C05447=1098.958,349.273,-87.589,179.031,19.110,152.319
C05448=1098.953,349.026,-87.554,179.028,19.106,152.319
C05449=1098.947,348.778,-87.521,179.025,19.103,152.319
C05450=1098.941,348.529,-87.486,179.022,19.099,152.318
C05451=1098.935,348.282,-87.452,179.019,19.095,152.318
C05452=1098.930,348.035,-87.418,179.016,19.092,152.318
C05453=1098.924,347.787,-87.385,179.013,19.089,152.318
C05454=1098.918,347.540,-87.351,179.010,19.084,152.317
C05455=1098.913,347.292,-87.316,179.007,19.081,152.317
C05456=1098.907,347.044,-87.283,179.003,19.078,152.317
C05457=1098.902,346.797,-87.249,179.000,19.074,152.316
C05458=1098.895,346.549,-87.214,178.998,19.071,152.316
C05459=1098.890,346.301,-87.181,178.994,19.067,152.316
C05460=1098.884,346.054,-87.147,178.992,19.064,152.316
C05461=1098.879,345.806,-87.112,178.988,19.060,152.315
C05462=1098.873,345.558,-87.079,178.985,19.057,152.315
C05463=1098.867,345.311,-87.045,178.982,19.053,152.315
C05464=1098.862,345.063,-87.011,178.979,19.050,152.314
C05465=1098.856,344.816,-86.977,178.976,19.046,152.314
C05466=1098.850,344.568,-86.944,178.973,19.043,152.314
C05467=1098.844,344.320,-86.910,178.969,19.039,152.314
C05468=1098.839,344.073,-86.877,178.966,19.036,152.313
C05469=1098.829,343.698,-86.825,178.962,19.031,152.313
C05470=1098.821,343.324,-86.774,178.957,19.026,152.313
C05471=1098.812,342.950,-86.724,178.952,19.021,152.312
C05472=1098.804,342.576,-86.673,178.947,19.015,152.312
C05473=1098.798,342.328,-86.640,178.945,19.012,152.312
C05474=1098.793,342.080,-86.606,178.941,19.008,152.311
C05475=1098.787,341.833,-86.572,178.938,19.006,152.311
C05476=1098.781,341.585,-86.539,178.935,19.003,152.311
C05477=1098.776,341.337,-86.505,178.932,18.999,152.311
C05478=1098.770,341.089,-86.472,178.929,18.996,152.311
C05479=1098.764,340.842,-86.438,178.925,18.992,152.310
C05480=1098.759,340.594,-86.404,178.923,18.989,152.310
C05481=1098.753,340.346,-86.371,178.920,18.986,152.310
C05482=1098.747,340.099,-86.338,178.916,18.982,152.310
C05483=1098.741,339.851,-86.305,178.913,18.979,152.310
C05484=1098.736,339.603,-86.271,178.910,18.975,152.309
C05485=1098.730,339.356,-86.237,178.907,18.972,152.309
C05486=1098.724,339.108,-86.204,178.904,18.970,152.309
C05487=1098.719,338.860,-86.171,178.901,18.966,152.309
C05488=1098.713,338.612,-86.137,178.898,18.963,152.308
C05489=1098.707,338.364,-86.105,178.895,18.960,152.308
C05490=1098.701,338.116,-86.071,178.891,18.956,152.308
C05491=1098.696,337.869,-86.038,178.888,18.953,152.308
C05492=1098.690,337.621,-86.004,178.885,18.950,152.308
C05493=1098.684,337.374,-85.971,178.882,18.947,152.308
C05494=1098.678,337.126,-85.938,178.879,18.944,152.307
C05495=1098.672,336.878,-85.904,178.875,18.940,152.307
C05496=1098.667,336.630,-85.871,178.872,18.937,152.307
C05497=1098.661,336.382,-85.838,178.870,18.934,152.307
C05498=1098.656,336.135,-85.805,178.866,18.931,152.307
C05499=1098.650,335.887,-85.772,178.863,18.928,152.306
C05500=1098.644,335.640,-85.739,178.860,18.925,152.306
C05501=1098.638,335.392,-85.706,178.856,18.921,152.306
C05502=1098.633,335.144,-85.673,178.853,18.919,152.306
C05503=1098.627,334.896,-85.641,178.851,18.915,152.306
C05504=1098.621,334.648,-85.607,178.848,18.913,152.306
C05505=1098.616,334.400,-85.574,178.844,18.909,152.305
C05506=1098.610,334.153,-85.542,178.841,18.906,152.305
C05507=1098.604,333.905,-85.508,178.838,18.903,152.305
C05508=1098.599,333.657,-85.475,178.834,18.900,152.305
C05509=1098.593,333.410,-85.442,178.831,18.897,152.305
C05510=1098.587,333.161,-85.410,178.829,18.894,152.305
C05511=1098.582,332.913,-85.376,178.825,18.891,152.305
C05512=1098.576,332.666,-85.344,178.822,18.888,152.304
C05513=1098.570,332.418,-85.311,178.819,18.885,152.304
C05514=1098.564,332.170,-85.278,178.815,18.881,152.304
C05515=1098.559,331.922,-85.245,178.812,18.879,152.304
C05516=1098.553,331.675,-85.212,178.809,18.876,152.304
C05517=1098.547,331.427,-85.179,178.806,18.873,152.304
C05518=1098.542,331.179,-85.147,178.803,18.870,152.304
C05519=1098.535,330.932,-85.115,178.800,18.867,152.304
C05520=1098.530,330.684,-85.081,178.797,18.864,152.303
C05521=1098.520,330.303,-85.031,178.791,18.859,152.303
C05522=1098.511,329.923,-84.981,178.787,18.855,152.303
C05523=1098.504,329.542,-84.932,178.781,18.851,152.303
C05524=1098.494,329.162,-84.881,178.777,18.846,152.303
C05525=1098.488,328.915,-84.849,178.774,18.844,152.303
C05526=1098.483,328.666,-84.816,178.770,18.840,152.303
C05527=1098.477,328.419,-84.784,178.767,18.838,152.303
C05528=1098.471,328.170,-84.752,178.764,18.835,152.303
C05529=1098.465,327.923,-84.719,178.761,18.832,152.302
C05530=1098.460,327.675,-84.687,178.757,18.829,152.302
C05531=1098.454,327.427,-84.654,178.754,18.826,152.302
C05532=1098.448,327.179,-84.622,178.751,18.823,152.302
C05533=1098.442,326.931,-84.589,178.748,18.821,152.302
C05534=1098.437,326.684,-84.557,178.745,18.818,152.302
C05535=1098.430,326.436,-84.524,178.742,18.815,152.302
C05536=1098.424,326.188,-84.492,178.738,18.812,152.302
C05537=1098.420,325.940,-84.460,178.735,18.810,152.302
C05538=1098.413,325.693,-84.427,178.732,18.807,152.302
C05539=1098.407,325.444,-84.395,178.729,18.803,152.302
C05540=1098.402,325.197,-84.363,178.726,18.801,152.302
C05541=1098.397,324.949,-84.330,178.723,18.798,152.301
C05542=1098.391,324.701,-84.298,178.720,18.795,152.301
C05543=1098.385,324.453,-84.266,178.717,18.793,152.301
C05544=1098.379,324.206,-84.234,178.713,18.790,152.301
C05545=1098.374,323.957,-84.201,178.710,18.787,152.301
C05546=1098.368,323.710,-84.169,178.707,18.784,152.301
C05547=1098.362,323.461,-84.137,178.704,18.781,152.301
C05548=1098.356,323.214,-84.105,178.701,18.779,152.301
C05549=1098.351,322.966,-84.073,178.698,18.776,152.301
C05550=1098.345,322.718,-84.040,178.693,18.773,152.301
C05551=1098.340,322.470,-84.009,178.690,18.770,152.301
C05552=1098.334,322.222,-83.977,178.687,18.768,152.301
C05553=1098.329,322.012,-83.950,178.684,18.765,152.301
C05554=1098.324,321.802,-83.922,178.682,18.763,152.301
C05555=1098.320,321.592,-83.895,178.679,18.760,152.301
C05556=1098.315,321.381,-83.868,178.677,18.759,152.301
C05557=1098.310,321.171,-83.841,178.674,18.756,152.301
C05558=1098.306,320.961,-83.814,178.671,18.754,152.300
C05559=1098.301,320.751,-83.787,178.668,18.752,152.301
C05560=1098.296,320.541,-83.760,178.666,18.749,152.300
C05561=1098.290,320.293,-83.728,178.663,18.747,152.300
C05562=1098.285,320.045,-83.696,178.659,18.744,152.300
C05563=1098.279,319.797,-83.664,178.656,18.741,152.300
C05564=1098.273,319.549,-83.632,178.653,18.738,152.300
C05565=1098.267,319.301,-83.600,178.650,18.736,152.300
C05566=1098.262,319.054,-83.568,178.647,18.733,152.300
C05567=1098.256,318.805,-83.536,178.644,18.731,152.300
C05568=1098.251,318.558,-83.505,178.640,18.728,152.300
C05569=1098.245,318.310,-83.473,178.637,18.725,152.300
C05570=1098.239,318.062,-83.441,178.634,18.722,152.300
C05571=1098.234,317.814,-83.408,178.630,18.720,152.300
C05572=1098.229,317.566,-83.377,178.627,18.717,152.300
C05573=1098.223,317.334,-83.348,178.624,18.715,152.300
C05574=1098.218,317.104,-83.318,178.621,18.712,152.300
C05575=1098.213,316.872,-83.288,178.618,18.709,152.300
C05576=1098.207,316.640,-83.259,178.616,18.708,152.300
C05577=1098.203,316.409,-83.229,178.613,18.705,152.300
C05578=1098.198,316.177,-83.200,178.609,18.703,152.300
C05579=1098.191,315.946,-83.170,178.606,18.700,152.300
C05580=1098.187,315.715,-83.141,178.603,18.698,152.300
C05581=1098.181,315.467,-83.109,178.600,18.695,152.300
C05582=1098.176,315.219,-83.077,178.597,18.692,152.300
C05583=1098.170,314.971,-83.045,178.594,18.690,152.300
C05584=1098.164,314.723,-83.014,178.591,18.687,152.300
C05585=1098.158,314.475,-82.983,178.587,18.685,152.300
C05586=1098.152,314.227,-82.951,178.584,18.682,152.300
C05587=1098.147,313.979,-82.920,178.581,18.680,152.300
C05588=1098.141,313.731,-82.889,178.578,18.678,152.300
C05589=1098.135,313.484,-82.857,178.574,18.675,152.300
C05590=1098.129,313.235,-82.826,178.571,18.673,152.300
C05591=1098.123,312.988,-82.795,178.568,18.670,152.300
C05592=1098.117,312.740,-82.763,178.564,18.668,152.300
C05593=1098.112,312.492,-82.732,178.561,18.665,152.300
C05594=1098.106,312.244,-82.700,178.558,18.663,152.300
C05595=1098.100,311.995,-82.669,178.555,18.661,152.300
C05596=1098.095,311.748,-82.638,178.552,18.658,152.300
C05597=1098.089,311.499,-82.607,178.548,18.656,152.300
C05598=1098.083,311.252,-82.575,178.545,18.653,152.300
C05599=1098.077,311.004,-82.544,178.542,18.651,152.300
C05600=1098.072,310.756,-82.513,178.539,18.649,152.300
C05601=1098.066,310.508,-82.481,178.535,18.646,152.300
C05602=1098.060,310.260,-82.451,178.532,18.644,152.300
C05603=1098.055,310.012,-82.420,178.528,18.641,152.300
C05604=1098.048,309.765,-82.389,178.525,18.639,152.300
C05605=1098.043,309.516,-82.357,178.522,18.636,152.300
C05606=1098.037,309.268,-82.326,178.519,18.634,152.301
C05607=1098.032,309.020,-82.295,178.515,18.632,152.301
C05608=1098.026,308.773,-82.264,178.512,18.629,152.301
C05609=1098.020,308.524,-82.233,178.509,18.627,152.301
C05610=1098.015,308.276,-82.202,178.506,18.624,152.301
C05611=1098.009,308.029,-82.171,178.503,18.622,152.301
C05612=1098.003,307.780,-82.140,178.499,18.620,152.301
C05613=1097.997,307.532,-82.109,178.496,18.617,152.301
C05614=1097.992,307.285,-82.078,178.493,18.615,152.301
C05615=1097.986,307.037,-82.047,178.490,18.613,152.301
C05616=1097.980,306.788,-82.016,178.486,18.610,152.301
C05617=1097.974,306.540,-81.986,178.483,18.608,152.301
C05618=1097.969,306.293,-81.954,178.480,18.606,152.301
C05619=1097.963,306.045,-81.924,178.477,18.604,152.301
C05620=1097.958,305.797,-81.893,178.473,18.601,152.301
C05621=1097.952,305.548,-81.862,178.470,18.599,152.301
C05622=1097.946,305.301,-81.830,178.467,18.597,152.301
C05623=1097.941,305.053,-81.800,178.464,18.594,152.301
C05624=1097.935,304.805,-81.769,178.460,18.592,152.302
C05625=1097.930,304.557,-81.739,178.457,18.590,152.302
C05626=1097.924,304.308,-81.707,178.453,18.587,152.302
C05627=1097.918,304.060,-81.677,178.450,18.585,152.302
C05628=1097.912,303.813,-81.647,178.447,18.582,152.302
C05629=1097.904,303.428,-81.598,178.442,18.579,152.302
C05630=1097.895,303.043,-81.551,178.437,18.575,152.302
C05631=1097.887,302.658,-81.503,178.432,18.572,152.302
C05632=1097.878,302.274,-81.455,178.427,18.568,152.302
C05633=1097.872,302.026,-81.425,178.424,18.566,152.302
C05634=1097.867,301.778,-81.394,178.421,18.564,152.302
C05635=1097.861,301.530,-81.364,178.417,18.562,152.302
C05636=1097.855,301.282,-81.334,178.414,18.559,152.302
C05637=1097.850,301.034,-81.303,178.411,18.557,152.303
C05638=1097.845,300.786,-81.273,178.408,18.555,152.303
C05639=1097.839,300.538,-81.242,178.404,18.552,152.303
C05640=1097.834,300.290,-81.211,178.401,18.550,152.303
C05641=1097.827,300.041,-81.181,178.398,18.548,152.303
C05642=1097.821,299.793,-81.150,178.395,18.545,152.303
C05643=1097.816,299.545,-81.119,178.391,18.543,152.303
C05644=1097.811,299.298,-81.089,178.388,18.541,152.303
C05645=1097.805,299.049,-81.059,178.385,18.539,152.303
C05646=1097.800,298.801,-81.028,178.381,18.537,152.303
C05647=1097.794,298.553,-80.998,178.378,18.534,152.303
C05648=1097.788,298.305,-80.968,178.375,18.532,152.303
C05649=1097.782,298.057,-80.937,178.372,18.530,152.303
C05650=1097.778,297.809,-80.907,178.368,18.527,152.304
C05651=1097.772,297.561,-80.877,178.365,18.526,152.304
C05652=1097.766,297.313,-80.846,178.362,18.523,152.304
C05653=1097.761,297.065,-80.817,178.358,18.521,152.304
C05654=1097.755,296.817,-80.787,178.355,18.519,152.304
C05655=1097.749,296.569,-80.756,178.352,18.517,152.304
C05656=1097.743,296.321,-80.726,178.348,18.515,152.304
C05657=1097.738,296.073,-80.696,178.345,18.512,152.304
C05658=1097.732,295.825,-80.666,178.342,18.510,152.305
C05659=1097.727,295.576,-80.636,178.338,18.508,152.305
C05660=1097.721,295.328,-80.605,178.335,18.506,152.305
C05661=1097.715,295.081,-80.575,178.332,18.504,152.305
C05662=1097.710,294.832,-80.545,178.328,18.502,152.305
C05663=1097.704,294.584,-80.515,178.325,18.499,152.305
C05664=1097.699,294.336,-80.485,178.322,18.498,152.305
C05665=1097.693,294.088,-80.455,178.319,18.496,152.305
C05666=1097.687,293.840,-80.425,178.316,18.494,152.306
C05667=1097.681,293.592,-80.395,178.312,18.492,152.306
C05668=1097.676,293.344,-80.365,178.309,18.489,152.306
C05669=1097.670,293.095,-80.335,178.306,18.487,152.306
C05670=1097.665,292.847,-80.305,178.302,18.485,152.306
C05671=1097.659,292.599,-80.275,178.299,18.483,152.306
C05672=1097.652,292.351,-80.246,178.296,18.481,152.306
C05673=1097.647,292.103,-80.216,178.292,18.479,152.306
C05674=1097.641,291.855,-80.186,178.289,18.477,152.307
C05675=1097.635,291.607,-80.156,178.286,18.474,152.307
C05676=1097.630,291.359,-80.126,178.283,18.473,152.307
C05677=1097.625,291.111,-80.097,178.280,18.471,152.307
C05678=1097.619,290.863,-80.066,178.276,18.469,152.307
C05679=1097.614,290.615,-80.037,178.273,18.467,152.307
C05680=1097.608,290.366,-80.007,178.269,18.465,152.307
C05681=1097.600,289.996,-79.963,178.264,18.461,152.308
C05682=1097.590,289.625,-79.918,178.259,18.458,152.308
C05683=1097.582,289.254,-79.874,178.255,18.456,152.308
C05684=1097.574,288.883,-79.829,178.250,18.453,152.308
C05685=1097.568,288.635,-79.800,178.247,18.451,152.308
C05686=1097.562,288.386,-79.771,178.243,18.449,152.309
C05687=1097.557,288.139,-79.740,178.240,18.447,152.309
C05688=1097.551,287.890,-79.711,178.236,18.445,152.309
C05689=1097.545,287.642,-79.682,178.233,18.443,152.309
C05690=1097.539,287.394,-79.652,178.230,18.441,152.309
C05691=1097.534,287.145,-79.622,178.227,18.439,152.309
C05692=1097.528,286.898,-79.594,178.224,18.437,152.310
C05693=1097.522,286.650,-79.563,178.220,18.435,152.310
C05694=1097.517,286.402,-79.534,178.217,18.433,152.310
C05695=1097.511,286.153,-79.504,178.213,18.431,152.310
C05696=1097.505,285.905,-79.475,178.210,18.429,152.310
C05697=1097.500,285.657,-79.445,178.207,18.427,152.310
C05698=1097.495,285.409,-79.416,178.204,18.425,152.311
C05699=1097.488,285.161,-79.387,178.200,18.424,152.311
C05700=1097.483,284.912,-79.357,178.197,18.421,152.311
C05701=1097.477,284.664,-79.328,178.194,18.419,152.311
C05702=1097.471,284.416,-79.299,178.190,18.418,152.311
C05703=1097.466,284.168,-79.269,178.187,18.415,152.311
C05704=1097.461,283.919,-79.240,178.183,18.413,152.312
C05705=1097.455,283.671,-79.211,178.181,18.412,152.312
C05706=1097.449,283.423,-79.181,178.177,18.410,152.312
C05707=1097.443,283.175,-79.152,178.174,18.408,152.312
C05708=1097.438,282.927,-79.123,178.171,18.406,152.312
C05709=1097.432,282.679,-79.093,178.167,18.404,152.312
C05710=1097.426,282.430,-79.065,178.164,18.402,152.313
C05711=1097.422,282.182,-79.036,178.161,18.400,152.313
C05712=1097.415,281.934,-79.007,178.158,18.398,152.313
C05713=1097.410,281.685,-78.977,178.154,18.397,152.313
C05714=1097.405,281.438,-78.948,178.151,18.394,152.313
C05715=1097.399,281.190,-78.919,178.147,18.392,152.313
C05716=1097.393,280.941,-78.890,178.144,18.391,152.314
C05717=1097.387,280.692,-78.861,178.142,18.389,152.314
C05718=1097.382,280.445,-78.831,178.138,18.387,152.314
C05719=1097.376,280.197,-78.802,178.134,18.385,152.314
C05720=1097.370,279.948,-78.774,178.131,18.383,152.314
C05721=1097.365,279.699,-78.744,178.127,18.381,152.315
C05722=1097.359,279.452,-78.716,178.125,18.380,152.315
C05723=1097.353,279.203,-78.686,178.122,18.378,152.315
C05724=1097.347,278.955,-78.658,178.118,18.376,152.315
C05725=1097.343,278.707,-78.628,178.115,18.374,152.315
C05726=1097.336,278.459,-78.599,178.111,18.372,152.316
C05727=1097.330,278.210,-78.571,178.109,18.371,152.316
C05728=1097.325,277.962,-78.542,178.105,18.369,152.316
C05729=1097.319,277.714,-78.513,178.102,18.367,152.316
C05730=1097.314,277.465,-78.484,178.098,18.365,152.316
C05731=1097.308,277.218,-78.455,178.095,18.363,152.316
C05732=1097.302,276.969,-78.427,178.092,18.361,152.317
C05733=1097.294,276.607,-78.385,178.087,18.359,152.317
C05734=1097.286,276.247,-78.343,178.082,18.356,152.317
C05735=1097.278,275.884,-78.301,178.077,18.353,152.318
C05736=1097.270,275.523,-78.259,178.072,18.350,152.318
C05737=1097.264,275.274,-78.230,178.069,18.349,152.318
C05738=1097.258,275.026,-78.201,178.066,18.347,152.318
C05739=1097.253,274.778,-78.173,178.062,18.345,152.319
C05740=1097.247,274.530,-78.144,178.059,18.344,152.319
C05741=1097.242,274.282,-78.116,178.056,18.342,152.319
C05742=1097.236,274.034,-78.087,178.053,18.340,152.319
C05743=1097.230,273.786,-78.059,178.049,18.338,152.319
C05744=1097.224,273.537,-78.030,178.046,18.336,152.320
C05745=1097.219,273.288,-78.001,178.042,18.334,152.320
C05746=1097.214,273.040,-77.973,178.040,18.333,152.320
C05747=1097.208,272.792,-77.944,178.036,18.331,152.320
C05748=1097.202,272.544,-77.916,178.033,18.330,152.321
C05749=1097.196,272.295,-77.887,178.029,18.328,152.321
C05750=1097.190,272.047,-77.859,178.026,18.326,152.321
C05751=1097.185,271.799,-77.830,178.023,18.325,152.321
C05752=1097.179,271.550,-77.801,178.019,18.323,152.321
C05753=1097.174,271.302,-77.774,178.016,18.321,152.322
C05754=1097.168,271.053,-77.745,178.014,18.319,152.322
C05755=1097.162,270.806,-77.717,178.010,18.317,152.322
C05756=1097.156,270.557,-77.688,178.006,18.315,152.322
C05757=1097.151,270.309,-77.660,178.003,18.314,152.322
C05758=1097.145,270.060,-77.632,178.000,18.312,152.323
C05759=1097.140,269.813,-77.603,177.997,18.310,152.323
C05760=1097.134,269.564,-77.574,177.993,18.309,152.323
C05761=1097.129,269.316,-77.546,177.990,18.307,152.323
C05762=1097.123,269.067,-77.518,177.987,18.305,152.324
C05763=1097.118,268.819,-77.490,177.984,18.304,152.324
C05764=1097.112,268.570,-77.462,177.980,18.302,152.324
C05765=1097.106,268.322,-77.434,177.977,18.300,152.324
C05766=1097.100,268.073,-77.405,177.974,18.299,152.324
C05767=1097.095,267.825,-77.378,177.970,18.297,152.325
C05768=1097.089,267.577,-77.348,177.967,18.295,152.325
C05769=1097.083,267.329,-77.321,177.964,18.294,152.325
C05770=1097.078,267.080,-77.292,177.961,18.292,152.325
C05771=1097.072,266.832,-77.264,177.957,18.290,152.326
C05772=1097.066,266.584,-77.236,177.953,18.289,152.326
C05773=1097.061,266.336,-77.208,177.951,18.287,152.326
C05774=1097.056,266.088,-77.180,177.947,18.285,152.326
C05775=1097.050,265.839,-77.152,177.944,18.284,152.327
C05776=1097.044,265.591,-77.124,177.940,18.282,152.327
C05777=1097.038,265.342,-77.097,177.937,18.280,152.327
C05778=1097.033,265.094,-77.069,177.934,18.279,152.327
C05779=1097.027,264.845,-77.040,177.930,18.277,152.328
C05780=1097.021,264.597,-77.012,177.928,18.276,152.328
C05781=1097.016,264.349,-76.985,177.924,18.274,152.328
C05782=1097.010,264.100,-76.956,177.921,18.272,152.328
C05783=1097.005,263.852,-76.928,177.917,18.270,152.329
C05784=1096.998,263.604,-76.900,177.914,18.269,152.329
C05785=1096.990,263.245,-76.860,177.909,18.266,152.329
C05786=1096.981,262.886,-76.820,177.904,18.264,152.330
C05787=1096.973,262.527,-76.780,177.900,18.262,152.330
C05788=1096.965,262.168,-76.740,177.895,18.259,152.330
C05789=1096.960,261.920,-76.713,177.892,18.258,152.331
C05790=1096.954,261.671,-76.684,177.888,18.257,152.331
C05791=1096.948,261.424,-76.657,177.885,18.255,152.331
C05792=1096.942,261.174,-76.629,177.882,18.253,152.331
C05793=1096.937,260.926,-76.601,177.879,18.252,152.332
C05794=1096.931,260.679,-76.574,177.875,18.250,152.332
C05795=1096.925,260.429,-76.546,177.872,18.249,152.332
C05796=1096.920,260.181,-76.518,177.869,18.247,152.333
C05797=1096.913,259.933,-76.491,177.865,18.245,152.333
C05798=1096.908,259.684,-76.463,177.862,18.244,152.333
C05799=1096.903,259.436,-76.435,177.859,18.243,152.333
C05800=1096.897,259.188,-76.409,177.855,18.241,152.334
C05801=1096.891,258.939,-76.380,177.852,18.239,152.334
C05802=1096.885,258.691,-76.352,177.849,18.238,152.334
C05803=1096.880,258.442,-76.326,177.845,18.236,152.334
C05804=1096.874,258.194,-76.297,177.842,18.235,152.335
C05805=1096.868,257.945,-76.271,177.839,18.233,152.335
C05806=1096.863,257.697,-76.243,177.835,18.231,152.335
C05807=1096.857,257.448,-76.215,177.833,18.230,152.335
C05808=1096.851,257.200,-76.188,177.829,18.229,152.336
C05809=1096.846,256.951,-76.161,177.825,18.227,152.336
C05810=1096.840,256.704,-76.133,177.823,18.226,152.336
C05811=1096.834,256.454,-76.106,177.819,18.224,152.336
C05812=1096.829,256.206,-76.078,177.816,18.222,152.337
C05813=1096.823,255.958,-76.051,177.813,18.221,152.337
C05814=1096.817,255.709,-76.023,177.809,18.219,152.337
C05815=1096.811,255.461,-75.996,177.806,18.217,152.338
C05816=1096.806,255.212,-75.969,177.803,18.216,152.338
C05817=1096.800,254.964,-75.942,177.799,18.215,152.338
C05818=1096.795,254.716,-75.914,177.796,18.213,152.338
C05819=1096.789,254.467,-75.887,177.793,18.212,152.339
C05820=1096.783,254.219,-75.859,177.789,18.210,152.339
C05821=1096.778,253.970,-75.833,177.787,18.208,152.339
C05822=1096.773,253.722,-75.805,177.783,18.207,152.340
C05823=1096.767,253.474,-75.778,177.779,18.205,152.340
C05824=1096.761,253.224,-75.750,177.777,18.204,152.340
C05825=1096.755,252.976,-75.724,177.773,18.202,152.340
C05826=1096.750,252.727,-75.697,177.770,18.200,152.340
C05827=1096.744,252.480,-75.669,177.767,18.199,152.341
C05828=1096.739,252.231,-75.642,177.763,18.198,152.341
C05829=1096.733,251.983,-75.615,177.760,18.196,152.341
C05830=1096.728,251.733,-75.588,177.757,18.195,152.342
C05831=1096.722,251.485,-75.561,177.753,18.193,152.342
C05832=1096.716,251.237,-75.533,177.751,18.192,152.342
C05833=1096.711,250.989,-75.506,177.747,18.190,152.342
C05834=1096.706,250.740,-75.479,177.744,18.188,152.343
C05835=1096.700,250.492,-75.453,177.741,18.187,152.343
C05836=1096.694,250.243,-75.426,177.737,18.186,152.343
C05837=1096.686,249.881,-75.386,177.733,18.183,152.344
C05838=1096.679,249.520,-75.347,177.727,18.181,152.344
C05839=1096.670,249.158,-75.308,177.723,18.179,152.344
C05840=1096.662,248.796,-75.268,177.718,18.177,152.345
C05841=1096.656,248.548,-75.241,177.715,18.175,152.345
C05842=1096.651,248.299,-75.214,177.712,18.174,152.345
C05843=1096.645,248.051,-75.187,177.708,18.172,152.346
C05844=1096.640,247.803,-75.161,177.706,18.170,152.346
C05845=1096.635,247.554,-75.134,177.702,18.169,152.346
C05846=1096.629,247.306,-75.107,177.698,18.167,152.346
C05847=1096.623,247.057,-75.080,177.696,18.166,152.347
C05848=1096.618,246.808,-75.054,177.692,18.165,152.347
C05849=1096.612,246.559,-75.027,177.689,18.163,152.347
C05850=1096.607,246.311,-75.000,177.686,18.161,152.348
C05851=1096.601,246.063,-74.974,177.682,18.160,152.348
C05852=1096.595,245.814,-74.947,177.679,18.159,152.348
C05853=1096.590,245.566,-74.920,177.676,18.157,152.348
C05854=1096.584,245.317,-74.893,177.673,18.156,152.349
C05855=1096.579,245.069,-74.867,177.669,18.154,152.349
C05856=1096.573,244.821,-74.840,177.666,18.153,152.349
C05857=1096.567,244.572,-74.814,177.663,18.151,152.350
C05858=1096.562,244.323,-74.787,177.659,18.150,152.350
C05859=1096.557,244.075,-74.760,177.657,18.149,152.350
C05860=1096.551,243.826,-74.733,177.653,18.147,152.350
C05861=1096.545,243.577,-74.707,177.650,18.146,152.351
C05862=1096.540,243.329,-74.681,177.647,18.144,152.351
C05863=1096.534,243.081,-74.654,177.643,18.142,152.351
C05864=1096.528,242.832,-74.628,177.640,18.141,152.352
C05865=1096.523,242.583,-74.602,177.637,18.140,152.352
C05866=1096.517,242.335,-74.575,177.634,18.139,152.352
C05867=1096.511,242.087,-74.548,177.630,18.137,152.353
C05868=1096.505,241.838,-74.522,177.627,18.136,152.353
C05869=1096.500,241.589,-74.496,177.624,18.134,152.353
C05870=1096.494,241.341,-74.469,177.620,18.133,152.353
C05871=1096.488,241.092,-74.443,177.617,18.132,152.354
C05872=1096.483,240.844,-74.417,177.614,18.130,152.354
C05873=1096.477,240.595,-74.390,177.611,18.129,152.354
C05874=1096.471,240.346,-74.364,177.607,18.127,152.355
C05875=1096.466,240.098,-74.337,177.604,18.126,152.355
C05876=1096.460,239.849,-74.311,177.601,18.125,152.355
C05877=1096.454,239.600,-74.285,177.598,18.123,152.356
C05878=1096.449,239.352,-74.258,177.594,18.122,152.356
C05879=1096.443,239.103,-74.232,177.591,18.120,152.356
C05880=1096.437,238.855,-74.205,177.588,18.119,152.356
C05881=1096.432,238.606,-74.180,177.584,18.118,152.357
C05882=1096.426,238.357,-74.153,177.581,18.116,152.357
C05883=1096.421,238.108,-74.127,177.578,18.115,152.357
C05884=1096.415,237.860,-74.100,177.575,18.114,152.358
C05885=1096.410,237.612,-74.075,177.571,18.112,152.358
C05886=1096.404,237.364,-74.049,177.568,18.111,152.358
C05887=1096.398,237.115,-74.023,177.565,18.109,152.359
C05888=1096.393,236.866,-73.997,177.562,18.108,152.359
C05889=1096.384,236.498,-73.958,177.557,18.106,152.359
C05890=1096.376,236.129,-73.919,177.552,18.104,152.360
C05891=1096.368,235.760,-73.881,177.547,18.102,152.360
C05892=1096.359,235.392,-73.842,177.543,18.100,152.361
C05893=1096.354,235.143,-73.816,177.539,18.098,152.361
C05894=1096.349,234.895,-73.790,177.536,18.097,152.361
C05895=1096.343,234.646,-73.764,177.533,18.096,152.362
C05896=1096.337,234.397,-73.738,177.530,18.095,152.362
C05897=1096.331,234.149,-73.712,177.526,18.093,152.362
C05898=1096.326,233.900,-73.686,177.524,18.092,152.362
C05899=1096.320,233.651,-73.660,177.520,18.090,152.363
C05900=1096.315,233.403,-73.634,177.517,18.089,152.363
C05901=1096.309,233.155,-73.608,177.513,18.088,152.363
C05902=1096.303,232.906,-73.582,177.511,18.086,152.364
C05903=1096.298,232.657,-73.556,177.507,18.085,152.364
C05904=1096.292,232.408,-73.531,177.504,18.084,152.364
C05905=1096.287,232.160,-73.506,177.500,18.082,152.365
C05906=1096.281,231.911,-73.479,177.498,18.081,152.365
C05907=1096.276,231.662,-73.453,177.494,18.079,152.365
C05908=1096.269,231.414,-73.428,177.491,18.078,152.366
C05909=1096.265,231.165,-73.402,177.488,18.077,152.366
C05910=1096.259,230.916,-73.376,177.485,18.076,152.366
C05911=1096.253,230.668,-73.351,177.481,18.074,152.367
C05912=1096.247,230.419,-73.325,177.478,18.073,152.367
C05913=1096.243,230.171,-73.299,177.475,18.071,152.367
C05914=1096.236,229.922,-73.274,177.472,18.071,152.368
C05915=1096.231,229.674,-73.247,177.468,18.069,152.368
C05916=1096.224,229.425,-73.222,177.465,18.068,152.368
C05917=1096.220,229.177,-73.196,177.462,18.066,152.368
C05918=1096.213,228.928,-73.171,177.459,18.065,152.369
C05919=1096.208,228.679,-73.145,177.455,18.064,152.369
C05920=1096.202,228.430,-73.120,177.452,18.063,152.369
C05921=1096.197,228.182,-73.094,177.449,18.061,152.370
C05922=1096.191,227.933,-73.069,177.446,18.060,152.370
C05923=1096.185,227.684,-73.043,177.442,18.058,152.370
C05924=1096.179,227.435,-73.018,177.439,18.057,152.371
C05925=1096.174,227.187,-72.993,177.437,18.056,152.371
C05926=1096.168,226.938,-72.967,177.433,18.055,152.371
C05927=1096.163,226.689,-72.942,177.430,18.054,152.372
C05928=1096.157,226.441,-72.917,177.426,18.052,152.372
C05929=1096.152,226.192,-72.891,177.424,18.051,152.372
C05930=1096.145,225.943,-72.865,177.420,18.050,152.373
C05931=1096.141,225.695,-72.840,177.417,18.048,152.373
C05932=1096.134,225.447,-72.814,177.413,18.047,152.373
C05933=1096.129,225.197,-72.789,177.411,18.046,152.374
C05934=1096.124,224.949,-72.764,177.407,18.044,152.374
C05935=1096.118,224.700,-72.738,177.404,18.043,152.374
C05936=1096.113,224.452,-72.713,177.400,18.042,152.375
C05937=1096.106,224.203,-72.688,177.398,18.041,152.375
C05938=1096.101,223.954,-72.663,177.395,18.040,152.375
C05939=1096.096,223.706,-72.638,177.391,18.038,152.376
C05940=1096.090,223.457,-72.612,177.388,18.037,152.376
C05941=1096.082,223.080,-72.574,177.383,18.035,152.376
C05942=1096.073,222.702,-72.536,177.378,18.033,152.377
C05943=1096.064,222.326,-72.498,177.373,18.031,152.377
C05944=1096.056,221.948,-72.459,177.369,18.029,152.378
C05945=1096.051,221.700,-72.434,177.365,18.027,152.378
C05946=1096.045,221.451,-72.410,177.362,18.027,152.378
C05947=1096.039,221.202,-72.384,177.359,18.026,152.379
C05948=1096.034,220.954,-72.359,177.356,18.024,152.379
C05949=1096.028,220.705,-72.334,177.353,18.023,152.380
C05950=1096.022,220.457,-72.309,177.349,18.021,152.380
C05951=1096.017,220.207,-72.284,177.346,18.021,152.380
C05952=1096.011,219.959,-72.259,177.343,18.019,152.380
C05953=1096.005,219.710,-72.234,177.340,18.018,152.381
C05954=1095.999,219.461,-72.209,177.337,18.017,152.381
C05955=1095.994,219.213,-72.183,177.333,18.015,152.381
C05956=1095.988,218.964,-72.159,177.330,18.015,152.382
C05957=1095.983,218.716,-72.134,177.327,18.013,152.382
C05958=1095.977,218.466,-72.109,177.324,18.012,152.383
C05959=1095.971,218.218,-72.084,177.321,18.011,152.383
C05960=1095.965,217.969,-72.060,177.317,18.009,152.383
C05961=1095.961,217.720,-72.035,177.315,18.008,152.383
C05962=1095.955,217.472,-72.009,177.311,18.007,152.384
C05963=1095.949,217.223,-71.985,177.308,18.006,152.384
C05964=1095.943,216.974,-71.960,177.305,18.005,152.384
C05965=1095.938,216.726,-71.936,177.301,18.003,152.385
C05966=1095.932,216.477,-71.910,177.299,18.002,152.385
C05967=1095.927,216.228,-71.885,177.295,18.001,152.386
C05968=1095.921,215.979,-71.861,177.292,18.000,152.386
C05969=1095.916,215.731,-71.836,177.289,17.999,152.386
C05970=1095.910,215.482,-71.811,177.286,17.997,152.386
C05971=1095.904,215.233,-71.787,177.283,17.996,152.387
C05972=1095.899,214.985,-71.762,177.279,17.994,152.387
C05973=1095.893,214.736,-71.737,177.276,17.994,152.387
C05974=1095.888,214.487,-71.713,177.274,17.992,152.388
C05975=1095.881,214.239,-71.688,177.270,17.991,152.388
C05976=1095.877,213.990,-71.663,177.267,17.990,152.388
C05977=1095.871,213.740,-71.638,177.263,17.988,152.389
C05978=1095.866,213.492,-71.614,177.260,17.988,152.389
C05979=1095.860,213.244,-71.589,177.258,17.986,152.389
C05980=1095.854,212.995,-71.564,177.254,17.985,152.390
C05981=1095.849,212.746,-71.540,177.251,17.984,152.390
C05982=1095.843,212.497,-71.516,177.248,17.983,152.390
C05983=1095.838,212.248,-71.491,177.245,17.981,152.391
C05984=1095.832,212.000,-71.466,177.242,17.980,152.391
C05985=1095.826,211.751,-71.442,177.238,17.979,152.392
C05986=1095.821,211.502,-71.417,177.235,17.978,152.392
C05987=1095.814,211.253,-71.393,177.232,17.977,152.392
C05988=1095.809,211.005,-71.369,177.229,17.975,152.392
C05989=1095.804,210.756,-71.345,177.226,17.974,152.393
C05990=1095.798,210.507,-71.320,177.223,17.973,152.393
C05991=1095.792,210.258,-71.296,177.219,17.972,152.393
C05992=1095.787,210.010,-71.271,177.216,17.971,152.394
C05993=1095.778,209.636,-71.235,177.212,17.969,152.394
C05994=1095.770,209.263,-71.198,177.207,17.967,152.395
C05995=1095.761,208.890,-71.162,177.202,17.966,152.395
C05996=1095.753,208.516,-71.126,177.198,17.964,152.396
C05997=1095.730,207.502,-71.027,177.146,17.942,152.401
C05998=1095.724,207.253,-71.003,177.143,17.942,152.402
C05999=1095.718,207.005,-70.979,177.139,17.942,152.402
C06000=1095.713,206.756,-70.955,177.136,17.942,152.403
C06001=1095.708,206.507,-70.931,177.133,17.941,152.403
C06002=1095.702,206.259,-70.908,177.129,17.940,152.404
C06003=1095.696,206.010,-70.883,177.126,17.940,152.404
C06004=1095.690,205.761,-70.859,177.122,17.940,152.405
C06005=1095.685,205.512,-70.836,177.119,17.939,152.405
C06006=1095.680,205.263,-70.812,177.116,17.939,152.406
C06007=1095.674,205.015,-70.788,177.113,17.939,152.406
C06008=1095.668,204.765,-70.764,177.109,17.938,152.407
C06009=1095.663,204.517,-70.740,177.106,17.938,152.408
C06010=1095.657,204.268,-70.716,177.103,17.938,152.408
C06011=1095.652,204.019,-70.693,177.100,17.938,152.409
C06012=1095.646,203.771,-70.669,177.096,17.937,152.409
C06013=1095.641,203.522,-70.645,177.093,17.937,152.410
C06014=1095.635,203.272,-70.621,177.090,17.937,152.410
C06015=1095.629,203.024,-70.597,177.087,17.936,152.411
C06016=1095.624,202.776,-70.573,177.083,17.936,152.411
C06017=1095.618,202.527,-70.550,177.080,17.936,152.412
C06018=1095.613,202.278,-70.526,177.077,17.936,152.413
C06019=1095.607,202.029,-70.503,177.073,17.936,152.413
C06020=1095.600,201.780,-70.479,177.070,17.935,152.414
C06021=1095.595,201.531,-70.455,177.067,17.935,152.414
C06022=1095.589,201.283,-70.431,177.064,17.935,152.415
C06023=1095.584,201.033,-70.408,177.060,17.934,152.415
C06024=1095.578,200.785,-70.384,177.057,17.934,152.416
C06025=1095.572,200.536,-70.361,177.053,17.933,152.416
C06026=1095.567,200.287,-70.337,177.050,17.933,152.417
C06027=1095.561,200.038,-70.314,177.047,17.932,152.418
C06028=1095.555,199.790,-70.290,177.043,17.932,152.418
C06029=1095.550,199.541,-70.267,177.040,17.932,152.419
C06030=1095.544,199.292,-70.243,177.037,17.932,152.419
C06031=1095.539,199.043,-70.219,177.034,17.931,152.420
C06032=1095.533,198.795,-70.196,177.030,17.931,152.420
C06033=1095.526,198.545,-70.172,177.027,17.931,152.421
C06034=1095.521,198.296,-70.149,177.024,17.930,152.421
C06035=1095.515,198.048,-70.125,177.021,17.930,152.422
C06036=1095.510,197.799,-70.102,177.017,17.930,152.423
C06037=1095.505,197.550,-70.079,177.014,17.929,152.423
C06038=1095.499,197.301,-70.055,177.011,17.929,152.424
C06039=1095.493,197.053,-70.032,177.008,17.929,152.424
C06040=1095.488,196.803,-70.009,177.004,17.929,152.425
C06041=1095.482,196.555,-69.985,177.001,17.928,152.425
C06042=1095.476,196.306,-69.962,176.998,17.928,152.426
C06043=1095.470,196.057,-69.939,176.995,17.928,152.426
C06044=1095.465,195.809,-69.915,176.991,17.927,152.427
C06045=1095.459,195.560,-69.892,176.988,17.927,152.427
C06046=1095.454,195.311,-69.869,176.985,17.927,152.428
C06047=1095.449,195.062,-69.845,176.982,17.926,152.429
C06048=1095.443,194.813,-69.822,176.978,17.926,152.429
C06049=1095.436,194.564,-69.798,176.975,17.925,152.430
C06050=1095.431,194.315,-69.775,176.972,17.925,152.430
C06051=1095.426,194.066,-69.752,176.969,17.925,152.431
C06052=1095.420,193.817,-69.729,176.966,17.924,152.431
C06053=1095.414,193.569,-69.706,176.962,17.924,152.432
C06054=1095.409,193.320,-69.683,176.959,17.924,152.432
C06055=1095.404,193.071,-69.659,176.956,17.924,152.433
C06056=1095.398,192.822,-69.636,176.953,17.923,152.433
C06057=1095.392,192.573,-69.613,176.950,17.923,152.434
C06058=1095.385,192.299,-69.588,176.946,17.923,152.434
C06059=1095.379,192.023,-69.561,176.943,17.922,152.435
C06060=1095.374,191.749,-69.537,176.939,17.922,152.436
C06061=1095.368,191.474,-69.511,176.936,17.921,152.436
C06062=1095.362,191.225,-69.488,176.932,17.921,152.437
C06063=1095.356,190.976,-69.465,176.929,17.920,152.437
C06064=1095.350,190.727,-69.442,176.926,17.920,152.438
C06065=1095.345,190.478,-69.418,176.923,17.920,152.438
C06066=1095.340,190.229,-69.395,176.920,17.919,152.439
C06067=1095.334,189.980,-69.372,176.916,17.919,152.439
C06068=1095.328,189.731,-69.349,176.913,17.918,152.440
C06069=1095.323,189.483,-69.327,176.910,17.918,152.440
C06070=1095.317,189.234,-69.304,176.907,17.918,152.441
C06071=1095.312,188.985,-69.280,176.904,17.917,152.441
C06072=1095.307,188.736,-69.257,176.901,17.917,152.442
C06073=1095.301,188.487,-69.234,176.897,17.916,152.442
C06074=1095.295,188.238,-69.212,176.894,17.916,152.443
C06075=1095.289,187.989,-69.189,176.891,17.915,152.443
C06076=1095.284,187.741,-69.166,176.888,17.915,152.444
C06077=1095.279,187.492,-69.143,176.885,17.915,152.444
C06078=1095.274,187.242,-69.120,176.882,17.915,152.445
C06079=1095.268,186.993,-69.097,176.879,17.914,152.445
C06080=1095.262,186.745,-69.074,176.876,17.914,152.446
C06081=1095.257,186.496,-69.051,176.873,17.914,152.446
C06082=1095.252,186.247,-69.029,176.870,17.913,152.447
C06083=1095.246,185.999,-69.006,176.867,17.913,152.447
C06084=1095.240,185.749,-68.984,176.863,17.912,152.448
C06085=1095.235,185.500,-68.961,176.860,17.911,152.448
C06086=1095.229,185.251,-68.938,176.857,17.911,152.449
C06087=1095.224,185.003,-68.915,176.854,17.911,152.449
C06088=1095.218,184.754,-68.892,176.851,17.910,152.450
C06089=1095.213,184.505,-68.870,176.848,17.910,152.450
C06090=1095.207,184.256,-68.847,176.844,17.910,152.451
C06091=1095.200,184.007,-68.825,176.841,17.909,152.452
C06092=1095.195,183.758,-68.802,176.838,17.909,152.452
C06093=1095.189,183.509,-68.780,176.835,17.909,152.453
C06094=1095.184,183.260,-68.757,176.832,17.908,152.453
C06095=1095.178,183.011,-68.734,176.828,17.908,152.454
C06096=1095.172,182.763,-68.712,176.826,17.908,152.454
C06097=1095.167,182.514,-68.689,176.823,17.908,152.455
C06098=1095.161,182.265,-68.666,176.819,17.907,152.455
C06099=1095.155,182.016,-68.644,176.816,17.907,152.456
C06100=1095.149,181.767,-68.622,176.813,17.906,152.456
C06101=1095.143,181.518,-68.599,176.810,17.906,152.457
C06102=1095.137,181.269,-68.576,176.807,17.906,152.457
C06103=1095.133,181.020,-68.554,176.804,17.905,152.458
C06104=1095.126,180.771,-68.532,176.800,17.905,152.458
C06105=1095.121,180.522,-68.510,176.797,17.904,152.459
C06106=1095.115,180.273,-68.487,176.794,17.904,152.459
C06107=1095.109,180.024,-68.464,176.791,17.903,152.460
C06108=1095.104,179.776,-68.442,176.788,17.903,152.460
C06109=1095.098,179.527,-68.419,176.784,17.903,152.461
C06110=1095.093,179.277,-68.397,176.782,17.903,152.461
C06111=1095.086,179.029,-68.375,176.779,17.902,152.462
C06112=1095.081,178.780,-68.353,176.776,17.902,152.462
C06113=1095.076,178.531,-68.330,176.773,17.901,152.463
C06114=1095.069,178.282,-68.308,176.770,17.901,152.463
C06115=1095.064,178.033,-68.285,176.766,17.901,152.464
C06116=1095.058,177.783,-68.263,176.763,17.900,152.464
C06117=1095.052,177.535,-68.241,176.760,17.900,152.465
C06118=1095.047,177.286,-68.219,176.757,17.899,152.465
C06119=1095.041,177.037,-68.196,176.754,17.899,152.466
C06120=1095.036,176.788,-68.175,176.751,17.898,152.466
C06121=1095.030,176.539,-68.153,176.748,17.898,152.467
C06122=1095.024,176.264,-68.128,176.744,17.897,152.467
C06123=1095.018,175.989,-68.103,176.741,17.897,152.468
C06124=1095.011,175.713,-68.078,176.738,17.897,152.468
C06125=1095.005,175.438,-68.055,176.735,17.897,152.469
C06126=1094.999,175.190,-68.032,176.732,17.896,152.469
C06127=1094.994,174.940,-68.010,176.728,17.896,152.470
C06128=1094.988,174.691,-67.987,176.725,17.895,152.470
C06129=1094.983,174.443,-67.966,176.722,17.895,152.471
C06130=1094.977,174.193,-67.943,176.719,17.894,152.471
C06131=1094.971,173.944,-67.922,176.716,17.894,152.472
C06132=1094.966,173.696,-67.899,176.713,17.893,152.472
C06133=1094.960,173.447,-67.878,176.710,17.893,152.473
C06134=1094.954,173.197,-67.855,176.707,17.892,152.473
C06135=1094.949,172.949,-67.833,176.704,17.892,152.474
C06136=1094.943,172.700,-67.811,176.701,17.891,152.474
C06137=1094.938,172.450,-67.789,176.698,17.891,152.475
C06138=1094.932,172.202,-67.768,176.695,17.890,152.475
C06139=1094.926,171.953,-67.745,176.692,17.890,152.476
C06140=1094.921,171.704,-67.723,176.689,17.889,152.476
C06141=1094.915,171.455,-67.701,176.685,17.889,152.477
C06142=1094.909,171.205,-67.680,176.683,17.889,152.477
C06143=1094.904,170.957,-67.658,176.680,17.889,152.478
C06144=1094.898,170.707,-67.636,176.677,17.888,152.478
C06145=1094.893,170.459,-67.613,176.674,17.887,152.478
C06146=1094.888,170.210,-67.591,176.671,17.887,152.479
C06147=1094.882,169.961,-67.570,176.668,17.886,152.479
C06148=1094.877,169.712,-67.548,176.665,17.886,152.480
C06149=1094.871,169.463,-67.526,176.662,17.885,152.480
C06150=1094.866,169.214,-67.504,176.659,17.885,152.481
C06151=1094.860,168.964,-67.483,176.656,17.885,152.481
C06152=1094.855,168.716,-67.461,176.653,17.884,152.482
C06153=1094.849,168.466,-67.439,176.650,17.883,152.482
C06154=1094.843,168.218,-67.416,176.647,17.883,152.483
C06155=1094.837,167.969,-67.395,176.644,17.882,152.483
C06156=1094.832,167.720,-67.373,176.641,17.881,152.483
C06157=1094.826,167.471,-67.351,176.638,17.881,152.484
C06158=1094.822,167.222,-67.329,176.636,17.881,152.484
C06159=1094.815,166.973,-67.308,176.633,17.880,152.485
C06160=1094.810,166.725,-67.287,176.629,17.880,152.485
C06161=1094.804,166.475,-67.264,176.626,17.879,152.486
C06162=1094.799,166.227,-67.243,176.623,17.878,152.486
C06163=1094.793,165.977,-67.221,176.620,17.878,152.487
C06164=1094.788,165.728,-67.200,176.617,17.877,152.487
C06165=1094.783,165.479,-67.178,176.614,17.877,152.488
C06166=1094.777,165.230,-67.157,176.612,17.877,152.488
C06167=1094.772,164.981,-67.135,176.609,17.876,152.488
C06168=1094.766,164.732,-67.113,176.606,17.876,152.489
C06169=1094.761,164.483,-67.092,176.603,17.875,152.489
C06170=1094.755,164.234,-67.070,176.600,17.874,152.490
C06171=1094.750,163.985,-67.049,176.597,17.873,152.490
C06172=1094.745,163.736,-67.027,176.593,17.873,152.491
C06173=1094.739,163.487,-67.005,176.591,17.873,152.491
C06174=1094.733,163.238,-66.984,176.588,17.872,152.492
C06175=1094.728,162.989,-66.962,176.585,17.871,152.492
C06176=1094.722,162.740,-66.941,176.582,17.871,152.492
C06177=1094.718,162.491,-66.919,176.579,17.870,152.493
C06178=1094.711,162.242,-66.897,176.576,17.870,152.493
C06179=1094.706,161.993,-66.877,176.573,17.869,152.494
C06180=1094.701,161.743,-66.855,176.571,17.869,152.494
C06181=1094.695,161.495,-66.833,176.568,17.868,152.494
C06182=1094.690,161.246,-66.812,176.565,17.867,152.495
C06183=1094.684,160.997,-66.791,176.562,17.867,152.495
C06184=1094.679,160.748,-66.769,176.559,17.866,152.496
C06185=1094.673,160.499,-66.748,176.556,17.866,152.496
C06186=1094.666,160.224,-66.725,176.552,17.865,152.497
C06187=1094.660,159.948,-66.700,176.549,17.865,152.497
C06188=1094.654,159.673,-66.677,176.546,17.864,152.498
C06189=1094.647,159.396,-66.654,176.543,17.864,152.498
C06190=1094.643,159.147,-66.632,176.540,17.863,152.499
C06191=1094.636,158.898,-66.611,176.537,17.862,152.499
C06192=1094.631,158.649,-66.590,176.534,17.862,152.500
C06193=1094.625,158.400,-66.569,176.532,17.862,152.500
C06194=1094.619,158.151,-66.547,176.529,17.861,152.500
C06195=1094.614,157.902,-66.527,176.526,17.860,152.501
C06196=1094.608,157.653,-66.505,176.523,17.860,152.501
C06197=1094.603,157.404,-66.485,176.520,17.859,152.502
C06198=1094.597,157.155,-66.463,176.517,17.859,152.502
C06199=1094.592,156.906,-66.441,176.514,17.858,152.503
C06200=1094.587,156.657,-66.420,176.511,17.858,152.503
C06201=1094.581,156.408,-66.399,176.508,17.857,152.503
C06202=1094.575,156.159,-66.378,176.505,17.856,152.504
C06203=1094.570,155.910,-66.357,176.503,17.855,152.504
C06204=1094.564,155.661,-66.336,176.500,17.855,152.505
C06205=1094.558,155.412,-66.315,176.497,17.855,152.505
C06206=1094.553,155.163,-66.294,176.494,17.854,152.506
C06207=1094.547,154.913,-66.273,176.491,17.854,152.506
C06208=1094.542,154.664,-66.252,176.488,17.853,152.506
C06209=1094.536,154.416,-66.231,176.486,17.853,152.507
C06210=1094.530,154.166,-66.210,176.483,17.852,152.507
C06211=1094.525,153.917,-66.189,176.480,17.851,152.508
C06212=1094.519,153.668,-66.168,176.477,17.850,152.508
C06213=1094.514,153.420,-66.147,176.474,17.850,152.508
C06214=1094.508,153.170,-66.126,176.472,17.850,152.509
C06215=1094.502,152.921,-66.105,176.469,17.849,152.509
C06216=1094.497,152.672,-66.084,176.466,17.849,152.510
C06217=1094.490,152.423,-66.064,176.463,17.848,152.510
C06218=1094.485,152.174,-66.042,176.460,17.847,152.511
C06219=1094.480,151.925,-66.022,176.457,17.847,152.511
C06220=1094.473,151.676,-66.000,176.454,17.846,152.511
C06221=1094.468,151.427,-65.980,176.451,17.846,152.512
C06222=1094.463,151.178,-65.959,176.448,17.845,152.512
C06223=1094.457,150.929,-65.938,176.445,17.844,152.513
C06224=1094.452,150.679,-65.917,176.443,17.844,152.513
C06225=1094.446,150.430,-65.896,176.440,17.843,152.513
C06226=1094.441,150.182,-65.875,176.437,17.842,152.514
C06227=1094.435,149.933,-65.855,176.434,17.842,152.514
C06228=1094.429,149.683,-65.834,176.431,17.841,152.515
C06229=1094.424,149.434,-65.814,176.429,17.841,152.515
C06230=1094.418,149.186,-65.792,176.426,17.840,152.515
C06231=1094.413,148.936,-65.772,176.423,17.839,152.516
C06232=1094.408,148.687,-65.751,176.420,17.839,152.516
C06233=1094.402,148.437,-65.730,176.417,17.838,152.517
C06234=1094.395,148.189,-65.710,176.415,17.838,152.517
C06235=1094.390,147.940,-65.689,176.412,17.837,152.518
C06236=1094.385,147.691,-65.669,176.409,17.836,152.518
C06237=1094.379,147.441,-65.648,176.406,17.836,152.518
C06238=1094.373,147.192,-65.628,176.404,17.835,152.519
C06239=1094.367,146.944,-65.606,176.401,17.834,152.519
C06240=1094.362,146.695,-65.586,176.398,17.833,152.519
C06241=1094.356,146.445,-65.566,176.395,17.833,152.520
C06242=1094.350,146.196,-65.545,176.392,17.832,152.520
C06243=1094.345,145.947,-65.525,176.390,17.832,152.521
C06244=1094.340,145.698,-65.504,176.387,17.831,152.521
C06245=1094.334,145.449,-65.484,176.384,17.830,152.521
C06246=1094.328,145.200,-65.462,176.381,17.830,152.522
C06247=1094.322,144.951,-65.442,176.379,17.830,152.522
C06248=1094.316,144.702,-65.422,176.376,17.829,152.523
C06249=1094.311,144.453,-65.401,176.373,17.828,152.523
C06250=1094.305,144.177,-65.379,176.370,17.827,152.523
C06251=1094.299,143.901,-65.356,176.367,17.827,152.524
C06252=1094.293,143.625,-65.333,176.364,17.826,152.524
C06253=1094.287,143.350,-65.311,176.361,17.825,152.525
C06254=1094.281,143.100,-65.290,176.358,17.825,152.525
C06255=1094.275,142.851,-65.270,176.355,17.823,152.525
C06256=1094.270,142.602,-65.249,176.353,17.823,152.526
C06257=1094.264,142.353,-65.229,176.350,17.822,152.526
C06258=1094.258,142.104,-65.209,176.347,17.822,152.527
C06259=1094.253,141.855,-65.188,176.344,17.821,152.527
C06260=1094.248,141.606,-65.168,176.341,17.820,152.527
C06261=1094.242,141.357,-65.148,176.339,17.820,152.528
C06262=1094.237,141.108,-65.127,176.336,17.819,152.528
C06263=1094.230,140.858,-65.107,176.333,17.818,152.529
C06264=1094.225,140.609,-65.086,176.330,17.817,152.529
C06265=1094.220,140.359,-65.067,176.328,17.817,152.529
C06266=1094.214,140.111,-65.047,176.325,17.816,152.530
C06267=1094.209,139.861,-65.026,176.322,17.815,152.530
C06268=1094.203,139.613,-65.006,176.319,17.815,152.530
C06269=1094.197,139.363,-64.986,176.317,17.814,152.531
C06270=1094.191,139.115,-64.966,176.314,17.813,152.531
C06271=1094.186,138.866,-64.945,176.311,17.813,152.531
C06272=1094.180,138.617,-64.925,176.308,17.812,152.532
C06273=1094.175,138.367,-64.905,176.307,17.811,152.532
C06274=1094.168,138.117,-64.885,176.304,17.811,152.533
C06275=1094.163,137.868,-64.864,176.301,17.810,152.533
C06276=1094.157,137.619,-64.844,176.298,17.810,152.533
C06277=1094.152,137.370,-64.824,176.296,17.808,152.534
C06278=1094.146,137.121,-64.805,176.293,17.808,152.534
C06279=1094.140,136.872,-64.785,176.290,17.807,152.534
C06280=1094.135,136.623,-64.764,176.288,17.806,152.535
C06281=1094.129,136.374,-64.744,176.285,17.806,152.535
C06282=1094.124,136.124,-64.724,176.282,17.805,152.536
C06283=1094.118,135.876,-64.704,176.279,17.804,152.536
C06284=1094.113,135.627,-64.684,176.277,17.804,152.536
C06285=1094.107,135.378,-64.664,176.274,17.803,152.537
C06286=1094.101,135.128,-64.645,176.271,17.802,152.537
C06287=1094.096,134.879,-64.624,176.268,17.801,152.537
C06288=1094.090,134.630,-64.604,176.266,17.801,152.538
C06289=1094.085,134.381,-64.584,176.263,17.800,152.538
C06290=1094.079,134.132,-64.564,176.260,17.799,152.538
C06291=1094.073,133.883,-64.544,176.258,17.799,152.539
C06292=1094.068,133.633,-64.524,176.255,17.798,152.539
C06293=1094.062,133.384,-64.505,176.252,17.797,152.539
C06294=1094.056,133.136,-64.485,176.249,17.796,152.540
C06295=1094.051,132.886,-64.465,176.248,17.796,152.540
C06296=1094.045,132.637,-64.445,176.245,17.795,152.540
C06297=1094.040,132.387,-64.425,176.242,17.794,152.541
C06298=1094.034,132.138,-64.405,176.239,17.793,152.541
C06299=1094.028,131.889,-64.386,176.237,17.793,152.542
C06300=1094.022,131.640,-64.366,176.234,17.792,152.542
C06301=1094.016,131.391,-64.346,176.231,17.791,152.542
C06302=1094.012,131.142,-64.326,176.229,17.790,152.542
C06303=1094.006,130.893,-64.306,176.226,17.789,152.543
C06304=1094.000,130.643,-64.287,176.223,17.789,152.543
C06305=1093.994,130.395,-64.267,176.220,17.788,152.544
C06306=1093.988,130.145,-64.248,176.218,17.787,152.544
C06307=1093.982,129.896,-64.228,176.215,17.787,152.544
C06308=1093.977,129.647,-64.208,176.212,17.786,152.545
C06309=1093.971,129.398,-64.188,176.210,17.785,152.545
C06310=1093.966,129.148,-64.169,176.207,17.784,152.545
C06311=1093.960,128.900,-64.149,176.205,17.783,152.546
C06312=1093.954,128.650,-64.129,176.203,17.783,152.546
C06313=1093.948,128.401,-64.109,176.200,17.782,152.546
C06314=1093.942,128.125,-64.088,176.197,17.781,152.547
C06315=1093.936,127.849,-64.066,176.194,17.780,152.547
C06316=1093.930,127.573,-64.045,176.191,17.780,152.547
C06317=1093.923,127.298,-64.023,176.188,17.779,152.548
C06318=1093.918,127.048,-64.003,176.185,17.778,152.548
C06319=1093.912,126.799,-63.984,176.183,17.777,152.549
C06320=1093.906,126.550,-63.964,176.180,17.776,152.549
C06321=1093.900,126.301,-63.945,176.177,17.776,152.549
C06322=1093.894,126.052,-63.925,176.175,17.774,152.549
C06323=1093.889,125.802,-63.905,176.172,17.774,152.550
C06324=1093.884,125.553,-63.886,176.170,17.773,152.550
C06325=1093.878,125.304,-63.866,176.167,17.772,152.551
C06326=1093.873,125.055,-63.847,176.165,17.772,152.551
C06327=1093.867,124.806,-63.828,176.162,17.771,152.551
C06328=1093.861,124.556,-63.809,176.159,17.770,152.551
C06329=1093.855,124.307,-63.789,176.157,17.769,152.552
C06330=1093.850,124.058,-63.769,176.154,17.768,152.552
C06331=1093.845,123.809,-63.751,176.151,17.767,152.552
C06332=1093.839,123.560,-63.731,176.149,17.767,152.553
C06333=1093.833,123.311,-63.711,176.147,17.766,152.553
C06334=1093.827,123.061,-63.692,176.144,17.765,152.553
C06335=1093.821,122.812,-63.673,176.141,17.764,152.554
C06336=1093.816,122.563,-63.654,176.139,17.763,152.554
C06337=1093.810,122.314,-63.634,176.136,17.762,152.554
C06338=1093.805,122.065,-63.614,176.133,17.762,152.555
C06339=1093.800,121.815,-63.595,176.131,17.761,152.555
C06340=1093.794,121.566,-63.576,176.129,17.760,152.555
C06341=1093.788,121.316,-63.556,176.126,17.759,152.556
C06342=1093.783,121.068,-63.538,176.124,17.758,152.556
C06343=1093.777,120.819,-63.518,176.121,17.757,152.556
C06344=1093.772,120.569,-63.498,176.118,17.756,152.557
C06345=1093.766,120.320,-63.479,176.116,17.756,152.557
C06346=1093.761,120.071,-63.460,176.113,17.755,152.557
C06347=1093.755,119.822,-63.441,176.111,17.753,152.557
C06348=1093.749,119.572,-63.422,176.108,17.753,152.558
C06349=1093.744,119.323,-63.403,176.106,17.752,152.558
C06350=1093.739,119.074,-63.384,176.103,17.751,152.558
C06351=1093.733,118.825,-63.364,176.101,17.750,152.558
C06352=1093.727,118.575,-63.345,176.098,17.750,152.559
C06353=1093.721,118.326,-63.327,176.095,17.748,152.559
C06354=1093.716,118.078,-63.308,176.093,17.748,152.559
C06355=1093.710,117.829,-63.288,176.091,17.747,152.560
C06356=1093.704,117.579,-63.268,176.088,17.746,152.560
C06357=1093.699,117.331,-63.250,176.086,17.745,152.560
C06358=1093.693,117.081,-63.230,176.083,17.744,152.561
C06359=1093.688,116.831,-63.212,176.080,17.743,152.561
C06360=1093.682,116.582,-63.193,176.078,17.742,152.561
C06361=1093.677,116.333,-63.174,176.076,17.741,152.561
C06362=1093.671,116.083,-63.154,176.073,17.740,152.562
C06363=1093.666,115.834,-63.135,176.071,17.740,152.562
C06364=1093.661,115.585,-63.116,176.068,17.739,152.562
C06365=1093.655,115.336,-63.097,176.065,17.737,152.563
C06366=1093.649,115.086,-63.078,176.063,17.737,152.563
C06367=1093.644,114.838,-63.059,176.061,17.736,152.563
C06368=1093.639,114.588,-63.040,176.058,17.734,152.563
C06369=1093.632,114.339,-63.021,176.056,17.734,152.564
C06370=1093.627,114.090,-63.002,176.053,17.733,152.564
C06371=1093.621,113.841,-62.983,176.050,17.732,152.564
C06372=1093.616,113.591,-62.964,176.048,17.731,152.565
C06373=1093.610,113.343,-62.946,176.046,17.730,152.565
C06374=1093.604,113.093,-62.927,176.043,17.729,152.565
C06375=1093.599,112.844,-62.908,176.041,17.729,152.565
C06376=1093.594,112.595,-62.889,176.038,17.728,152.566
C06377=1093.587,112.346,-62.870,176.035,17.726,152.566
C06378=1093.581,112.069,-62.850,176.033,17.726,152.566
C06379=1093.575,111.793,-62.828,176.031,17.725,152.567
C06380=1093.569,111.517,-62.808,176.028,17.724,152.567
C06381=1093.563,111.242,-62.787,176.025,17.723,152.567
C06382=1093.557,110.992,-62.768,176.022,17.721,152.567
C06383=1093.551,110.743,-62.749,176.020,17.720,152.568
C06384=1093.546,110.494,-62.731,176.018,17.720,152.568
C06385=1093.540,110.244,-62.712,176.015,17.718,152.568
C06386=1093.534,109.995,-62.693,176.013,17.718,152.569
C06387=1093.529,109.746,-62.674,176.010,17.717,152.569
C06388=1093.523,109.497,-62.656,176.007,17.716,152.569
C06389=1093.518,109.248,-62.637,176.005,17.715,152.569
C06390=1093.512,108.998,-62.618,176.003,17.714,152.570
C06391=1093.506,108.749,-62.600,176.000,17.713,152.570
C06392=1093.501,108.500,-62.581,175.998,17.712,152.570
C06393=1093.494,108.251,-62.563,175.995,17.711,152.571
C06394=1093.489,108.001,-62.544,175.993,17.710,152.571
C06395=1093.484,107.752,-62.525,175.991,17.709,152.571
C06396=1093.477,107.503,-62.507,175.988,17.708,152.571
C06397=1093.473,107.254,-62.489,175.986,17.708,152.572
C06398=1093.466,107.005,-62.470,175.983,17.706,152.572
C06399=1093.460,106.755,-62.451,175.981,17.705,152.572
C06400=1093.455,106.506,-62.433,175.979,17.705,152.572
C06401=1093.449,106.257,-62.414,175.976,17.703,152.573
C06402=1093.444,106.007,-62.396,175.973,17.702,152.573
C06403=1093.438,105.758,-62.377,175.971,17.702,152.573
C06404=1093.433,105.509,-62.359,175.969,17.700,152.573
C06405=1093.427,105.260,-62.340,175.967,17.700,152.574
C06406=1093.422,105.011,-62.321,175.964,17.699,152.574
C06407=1093.416,104.761,-62.303,175.961,17.697,152.574
C06408=1093.410,104.512,-62.284,175.959,17.697,152.574
C06409=1093.404,104.263,-62.267,175.957,17.696,152.575
C06410=1093.399,104.013,-62.247,175.955,17.695,152.575
C06411=1093.393,103.764,-62.230,175.952,17.694,152.575
C06412=1093.388,103.515,-62.211,175.949,17.693,152.575
C06413=1093.382,103.266,-62.193,175.947,17.692,152.576
C06414=1093.376,103.016,-62.174,175.945,17.691,152.576
C06415=1093.371,102.767,-62.156,175.942,17.690,152.576
C06416=1093.365,102.517,-62.138,175.940,17.689,152.576
C06417=1093.360,102.269,-62.119,175.938,17.687,152.577
C06418=1093.354,102.019,-62.101,175.936,17.687,152.577
C06419=1093.348,101.770,-62.083,175.933,17.686,152.577
C06420=1093.343,101.520,-62.064,175.930,17.684,152.577
C06421=1093.337,101.272,-62.046,175.928,17.684,152.578
C06422=1093.332,101.022,-62.027,175.926,17.683,152.578
C06423=1093.326,100.773,-62.010,175.924,17.682,152.578
C06424=1093.320,100.524,-61.991,175.921,17.681,152.578
C06425=1093.315,100.274,-61.973,175.918,17.680,152.579
C06426=1093.309,100.025,-61.955,175.917,17.678,152.579
C06427=1093.303,99.776,-61.937,175.914,17.677,152.579
C06428=1093.298,99.526,-61.918,175.912,17.677,152.579
C06429=1093.292,99.277,-61.901,175.909,17.675,152.580
C06430=1093.286,99.028,-61.882,175.906,17.674,152.580
C06431=1093.281,98.779,-61.864,175.905,17.674,152.580
C06432=1093.276,98.530,-61.846,175.902,17.673,152.580
C06433=1093.269,98.280,-61.828,175.900,17.672,152.581
C06434=1093.264,98.031,-61.810,175.897,17.670,152.581
C06435=1093.258,97.781,-61.791,175.895,17.669,152.581
C06436=1093.252,97.533,-61.773,175.893,17.668,152.581
C06437=1093.246,97.283,-61.755,175.890,17.667,152.582
C06438=1093.241,97.034,-61.737,175.888,17.667,152.582
C06439=1093.235,96.784,-61.719,175.886,17.665,152.582
C06440=1093.230,96.536,-61.701,175.883,17.664,152.582
C06441=1093.223,96.286,-61.683,175.881,17.663,152.582
C06442=1093.218,96.010,-61.663,175.878,17.662,152.583
C06443=1093.212,95.735,-61.643,175.876,17.661,152.583
C06444=1093.206,95.458,-61.623,175.873,17.660,152.583
C06445=1093.199,95.182,-61.603,175.870,17.658,152.583
C06446=1093.193,94.933,-61.585,175.869,17.657,152.584
C06447=1093.188,94.684,-61.568,175.866,17.656,152.584
C06448=1093.182,94.434,-61.549,175.864,17.656,152.584
C06449=1093.176,94.185,-61.531,175.861,17.654,152.584
C06450=1093.171,93.936,-61.513,175.859,17.653,152.585
C06451=1093.165,93.686,-61.495,175.857,17.652,152.585
C06452=1093.160,93.437,-61.477,175.854,17.651,152.585
C06453=1093.155,93.188,-61.460,175.852,17.650,152.585
C06454=1093.148,92.938,-61.442,175.850,17.649,152.585
C06455=1093.143,92.689,-61.424,175.848,17.648,152.586
C06456=1093.137,92.440,-61.407,175.845,17.646,152.586
C06457=1093.132,92.190,-61.388,175.843,17.645,152.586
C06458=1093.126,91.941,-61.371,175.841,17.645,152.586
C06459=1093.121,91.692,-61.353,175.838,17.643,152.586
C06460=1093.115,91.443,-61.334,175.836,17.642,152.587
C06461=1093.109,91.194,-61.317,175.834,17.641,152.587
C06462=1093.104,90.945,-61.299,175.832,17.640,152.587
C06463=1093.098,90.695,-61.281,175.829,17.639,152.587
C06464=1093.093,90.446,-61.263,175.827,17.638,152.588
C06465=1093.086,90.196,-61.245,175.825,17.636,152.588
C06466=1093.081,89.947,-61.228,175.822,17.635,152.588
C06467=1093.075,89.698,-61.210,175.820,17.635,152.588
C06468=1093.069,89.448,-61.192,175.818,17.634,152.588
C06469=1093.064,89.199,-61.175,175.816,17.632,152.589
C06470=1093.058,88.950,-61.157,175.813,17.631,152.589
C06471=1093.052,88.700,-61.140,175.810,17.630,152.589
C06472=1093.047,88.451,-61.122,175.809,17.629,152.589
C06473=1093.041,88.202,-61.105,175.806,17.628,152.589
C06474=1093.035,87.952,-61.087,175.804,17.627,152.590
C06475=1093.030,87.703,-61.069,175.802,17.625,152.590
C06476=1093.024,87.454,-61.052,175.800,17.625,152.590
C06477=1093.018,87.204,-61.034,175.797,17.623,152.590
C06478=1093.013,86.955,-61.016,175.795,17.623,152.590
C06479=1093.007,86.706,-60.998,175.793,17.621,152.591
C06480=1093.001,86.456,-60.981,175.790,17.620,152.591
C06481=1092.995,86.208,-60.964,175.788,17.619,152.591
C06482=1092.990,85.958,-60.947,175.786,17.617,152.591
C06483=1092.984,85.709,-60.929,175.784,17.617,152.591
C06484=1092.978,85.459,-60.911,175.781,17.616,152.592
C06485=1092.972,85.210,-60.894,175.780,17.615,152.592
C06486=1092.967,84.961,-60.876,175.777,17.613,152.592
C06487=1092.962,84.711,-60.859,175.775,17.612,152.592
C06488=1092.956,84.462,-60.841,175.773,17.611,152.592
C06489=1092.950,84.213,-60.824,175.770,17.609,152.593
C06490=1092.944,83.964,-60.806,175.768,17.609,152.593
C06491=1092.939,83.715,-60.789,175.766,17.607,152.593
C06492=1092.933,83.464,-60.771,175.764,17.607,152.593
C06493=1092.928,83.215,-60.754,175.761,17.605,152.593
C06494=1092.922,82.966,-60.736,175.759,17.604,152.594
C06495=1092.917,82.717,-60.719,175.757,17.603,152.594
C06496=1092.911,82.467,-60.701,175.755,17.602,152.594
C06497=1092.905,82.218,-60.685,175.753,17.600,152.594
C06498=1092.899,81.969,-60.667,175.751,17.600,152.594
C06499=1092.894,81.719,-60.650,175.748,17.598,152.594
C06500=1092.888,81.470,-60.633,175.746,17.597,152.595
C06501=1092.883,81.221,-60.615,175.744,17.596,152.595
C06502=1092.877,80.971,-60.598,175.741,17.595,152.595
C06503=1092.871,80.722,-60.580,175.740,17.593,152.595
C06504=1092.866,80.473,-60.563,175.737,17.592,152.595
C06505=1092.861,80.223,-60.546,175.735,17.591,152.596
C06506=1092.854,79.948,-60.527,175.732,17.590,152.596
C06507=1092.848,79.672,-60.508,175.730,17.588,152.596
C06508=1092.842,79.396,-60.488,175.728,17.587,152.596
C06509=1092.835,79.119,-60.469,175.726,17.586,152.596
C06510=1092.830,78.870,-60.452,175.723,17.584,152.596
C06511=1092.824,78.621,-60.435,175.720,17.583,152.597
C06512=1092.818,78.372,-60.418,175.719,17.582,152.597
C06513=1092.813,78.123,-60.400,175.716,17.581,152.597
C06514=1092.807,77.873,-60.384,175.714,17.580,152.597
C06515=1092.801,77.623,-60.366,175.712,17.578,152.597
C06516=1092.795,77.374,-60.349,175.710,17.578,152.598
C06517=1092.790,77.125,-60.332,175.708,17.576,152.598
C06518=1092.785,76.875,-60.315,175.706,17.575,152.598
C06519=1092.778,76.627,-60.298,175.703,17.574,152.598
C06520=1092.773,76.377,-60.281,175.701,17.573,152.598
C06521=1092.768,76.128,-60.264,175.699,17.571,152.598
C06522=1092.761,75.878,-60.247,175.697,17.570,152.599
C06523=1092.755,75.629,-60.229,175.695,17.569,152.599
C06524=1092.750,75.379,-60.212,175.693,17.568,152.599
C06525=1092.744,75.131,-60.195,175.690,17.567,152.599
C06526=1092.739,74.881,-60.179,175.689,17.566,152.599
C06527=1092.733,74.632,-60.161,175.686,17.564,152.599
C06528=1092.727,74.382,-60.145,175.684,17.563,152.600
C06529=1092.722,74.133,-60.127,175.682,17.562,152.600
C06530=1092.716,73.883,-60.110,175.680,17.561,152.600
C06531=1092.710,73.634,-60.094,175.677,17.559,152.600
C06532=1092.704,73.385,-60.076,175.676,17.558,152.600
C06533=1092.699,73.135,-60.059,175.673,17.557,152.600
C06534=1092.693,72.886,-60.042,175.671,17.555,152.601
C06535=1092.688,72.637,-60.026,175.669,17.554,152.601
C06536=1092.683,72.387,-60.009,175.666,17.553,152.601
C06537=1092.676,72.138,-59.992,175.665,17.552,152.601
C06538=1092.671,71.889,-59.975,175.662,17.550,152.601
C06539=1092.665,71.639,-59.959,175.660,17.549,152.601
C06540=1092.660,71.390,-59.941,175.658,17.548,152.602
C06541=1092.654,71.141,-59.925,175.656,17.547,152.602
C06542=1092.648,70.891,-59.908,175.654,17.545,152.602
C06543=1092.642,70.641,-59.890,175.652,17.544,152.602
C06544=1092.636,70.392,-59.874,175.649,17.543,152.602
C06545=1092.631,70.142,-59.857,175.648,17.542,152.602
C06546=1092.625,69.894,-59.840,175.645,17.540,152.602
C06547=1092.620,69.644,-59.823,175.644,17.539,152.603
C06548=1092.614,69.395,-59.807,175.641,17.538,152.603
C06549=1092.609,69.145,-59.790,175.639,17.537,152.603
C06550=1092.602,68.896,-59.773,175.637,17.535,152.603
C06551=1092.597,68.647,-59.756,175.635,17.535,152.603
C06552=1092.591,68.397,-59.740,175.632,17.533,152.603
C06553=1092.586,68.148,-59.723,175.631,17.532,152.603
C06554=1092.580,67.899,-59.706,175.628,17.530,152.604
C06555=1092.574,67.649,-59.689,175.626,17.530,152.604
C06556=1092.569,67.400,-59.673,175.624,17.528,152.604
C06557=1092.563,67.150,-59.656,175.622,17.527,152.604
C06558=1092.557,66.901,-59.640,175.620,17.525,152.604
C06559=1092.551,66.652,-59.624,175.618,17.525,152.604
C06560=1092.546,66.403,-59.606,175.615,17.523,152.605
C06561=1092.540,66.153,-59.590,175.614,17.522,152.605
C06562=1092.535,65.904,-59.573,175.612,17.521,152.605
C06563=1092.529,65.654,-59.557,175.610,17.519,152.605
C06564=1092.523,65.405,-59.540,175.608,17.518,152.605
C06565=1092.518,65.155,-59.524,175.605,17.517,152.605
C06566=1092.512,64.906,-59.507,175.604,17.516,152.605
C06567=1092.506,64.657,-59.490,175.601,17.514,152.605
C06568=1092.500,64.407,-59.473,175.600,17.513,152.606
C06569=1092.494,64.158,-59.457,175.597,17.512,152.606
C06570=1092.486,63.793,-59.432,175.594,17.510,152.606
C06571=1092.478,63.428,-59.409,175.591,17.508,152.606
C06572=1092.469,63.063,-59.385,175.588,17.506,152.607
C06573=1092.460,62.698,-59.361,175.585,17.504,152.607
C06574=1092.455,62.448,-59.344,175.583,17.503,152.607
C06575=1092.449,62.199,-59.328,175.581,17.502,152.607
C06576=1092.443,61.949,-59.312,175.578,17.500,152.607
C06577=1092.437,61.700,-59.295,175.577,17.499,152.607
C06578=1092.431,61.451,-59.279,175.574,17.498,152.607
C06579=1092.426,61.201,-59.262,175.573,17.497,152.607
C06580=1092.420,60.952,-59.246,175.570,17.495,152.608
C06581=1092.414,60.702,-59.230,175.568,17.494,152.608
C06582=1092.408,60.453,-59.214,175.566,17.493,152.608
C06583=1092.402,60.204,-59.197,175.564,17.492,152.608
C06584=1092.397,59.955,-59.181,175.563,17.490,152.608
C06585=1092.392,59.705,-59.165,175.560,17.489,152.608
C06586=1092.386,59.456,-59.148,175.558,17.488,152.608
C06587=1092.380,59.207,-59.132,175.556,17.487,152.609
C06588=1092.374,58.957,-59.116,175.554,17.485,152.609
C06589=1092.368,58.708,-59.100,175.552,17.484,152.609
C06590=1092.363,58.458,-59.083,175.550,17.483,152.609
C06591=1092.357,58.208,-59.067,175.548,17.481,152.609
C06592=1092.351,57.959,-59.051,175.546,17.480,152.609
C06593=1092.345,57.710,-59.035,175.543,17.478,152.609
C06594=1092.339,57.460,-59.018,175.542,17.477,152.609
C06595=1092.333,57.211,-59.002,175.539,17.476,152.610
C06596=1092.328,56.962,-58.986,175.537,17.475,152.610
C06597=1092.322,56.713,-58.969,175.536,17.474,152.610
C06598=1092.317,56.463,-58.954,175.533,17.472,152.610
C06599=1092.311,56.213,-58.938,175.532,17.471,152.610
C06600=1092.305,55.964,-58.921,175.529,17.469,152.610
C06601=1092.299,55.715,-58.905,175.528,17.468,152.610
C06602=1092.293,55.465,-58.889,175.525,17.467,152.611
C06603=1092.287,55.215,-58.873,175.524,17.465,152.611
C06604=1092.282,54.967,-58.857,175.521,17.464,152.611
C06605=1092.277,54.717,-58.841,175.520,17.463,152.611
C06606=1092.271,54.468,-58.824,175.517,17.461,152.611
C06607=1092.265,54.218,-58.808,175.515,17.460,152.611
C06608=1092.259,53.968,-58.793,175.514,17.459,152.611
C06609=1092.253,53.719,-58.776,175.511,17.457,152.611
C06610=1092.248,53.470,-58.760,175.510,17.456,152.611
C06611=1092.242,53.220,-58.745,175.507,17.454,152.612
C06612=1092.236,52.971,-58.729,175.506,17.453,152.612
C06613=1092.230,52.722,-58.712,175.503,17.452,152.612
C06614=1092.224,52.472,-58.696,175.502,17.450,152.612
C06615=1092.219,52.223,-58.681,175.499,17.449,152.612
C06616=1092.214,51.973,-58.664,175.497,17.448,152.612
C06617=1092.208,51.724,-58.648,175.496,17.447,152.612
C06618=1092.203,51.474,-58.632,175.493,17.445,152.612
C06619=1092.197,51.225,-58.616,175.492,17.444,152.612
C06620=1092.191,50.976,-58.600,175.489,17.442,152.613
C06621=1092.186,50.726,-58.585,175.488,17.441,152.613
C06622=1092.180,50.477,-58.568,175.485,17.439,152.613
C06623=1092.174,50.227,-58.553,175.484,17.438,152.613
C06624=1092.169,49.978,-58.537,175.482,17.437,152.613
C06625=1092.163,49.729,-58.521,175.479,17.435,152.613
C06626=1092.153,49.319,-58.495,175.476,17.433,152.613
C06627=1092.144,48.909,-58.469,175.473,17.431,152.613
C06628=1092.135,48.499,-58.442,175.470,17.428,152.613
C06629=1092.126,48.090,-58.417,175.467,17.426,152.614
C06630=1092.119,47.813,-58.399,175.464,17.424,152.614
C06631=1092.113,47.537,-58.382,175.463,17.423,152.614
C06632=1092.107,47.260,-58.364,175.460,17.422,152.614
C06633=1092.101,46.984,-58.347,175.458,17.420,152.614
C06634=1092.095,46.735,-58.331,175.456,17.419,152.614
C06635=1092.089,46.485,-58.315,175.454,17.417,152.614
C06636=1092.084,46.236,-58.299,175.452,17.416,152.614
C06637=1092.078,45.987,-58.284,175.451,17.415,152.614
C06638=1092.072,45.737,-58.268,175.448,17.413,152.615
C06639=1092.067,45.488,-58.253,175.446,17.412,152.615
C06640=1092.061,45.239,-58.236,175.444,17.410,152.615
C06641=1092.056,44.989,-58.221,175.442,17.409,152.615
C06642=1092.050,44.740,-58.205,175.440,17.407,152.615
C06643=1092.045,44.490,-58.189,175.439,17.406,152.615
C06644=1092.039,44.240,-58.174,175.437,17.405,152.615
C06645=1092.034,43.991,-58.158,175.434,17.403,152.615
C06646=1092.028,43.741,-58.142,175.433,17.402,152.615
C06647=1092.021,43.492,-58.127,175.430,17.400,152.615
C06648=1092.016,43.243,-58.111,175.429,17.399,152.616
C06649=1092.011,42.993,-58.096,175.427,17.398,152.615
C06650=1092.005,42.744,-58.080,175.425,17.396,152.616
C06651=1092.000,42.494,-58.065,175.423,17.395,152.616
C06652=1091.993,42.245,-58.050,175.421,17.393,152.616
C06653=1091.987,41.995,-58.033,175.419,17.392,152.616
C06654=1091.982,41.746,-58.018,175.418,17.391,152.616
C06655=1091.977,41.496,-58.003,175.415,17.389,152.616
C06656=1091.971,41.247,-57.986,175.414,17.388,152.616
C06657=1091.965,40.998,-57.972,175.411,17.386,152.616
C06658=1091.959,40.748,-57.956,175.410,17.385,152.616
C06659=1091.953,40.499,-57.940,175.408,17.384,152.616
C06660=1091.948,40.249,-57.925,175.406,17.382,152.617
C06661=1091.942,40.000,-57.910,175.404,17.381,152.617
C06662=1091.937,39.751,-57.894,175.402,17.379,152.617
C06663=1091.931,39.501,-57.878,175.400,17.378,152.617
C06664=1091.925,39.251,-57.863,175.399,17.377,152.617
C06665=1091.920,39.002,-57.848,175.396,17.375,152.617
C06666=1091.914,38.753,-57.832,175.394,17.374,152.617
C06667=1091.909,38.504,-57.817,175.392,17.372,152.617
C06668=1091.903,38.254,-57.801,175.391,17.371,152.617
C06669=1091.897,38.004,-57.786,175.389,17.369,152.617
C06670=1091.892,37.755,-57.771,175.387,17.368,152.617
C06671=1091.886,37.505,-57.755,175.385,17.367,152.617
C06672=1091.879,37.256,-57.740,175.383,17.365,152.617
C06673=1091.874,37.006,-57.725,175.381,17.363,152.618
C06674=1091.868,36.757,-57.710,175.379,17.362,152.618
C06675=1091.863,36.507,-57.695,175.377,17.361,152.618
C06676=1091.856,36.258,-57.679,175.375,17.360,152.618
C06677=1091.850,36.008,-57.663,175.373,17.358,152.618
C06678=1091.845,35.759,-57.648,175.372,17.356,152.618
C06679=1091.839,35.510,-57.633,175.370,17.355,152.618
C06680=1091.834,35.260,-57.618,175.367,17.353,152.618
C06681=1091.828,35.011,-57.603,175.366,17.352,152.618
C06682=1091.822,34.761,-57.588,175.364,17.351,152.618
C06683=1091.816,34.512,-57.573,175.362,17.349,152.618
C06684=1091.810,34.262,-57.557,175.360,17.348,152.618
C06685=1091.805,34.013,-57.542,175.358,17.346,152.619
C06686=1091.799,33.763,-57.527,175.356,17.345,152.619
C06687=1091.794,33.514,-57.512,175.355,17.344,152.619
C06688=1091.787,33.264,-57.497,175.352,17.342,152.619
C06689=1091.782,33.015,-57.481,175.351,17.341,152.619
C06690=1091.776,32.766,-57.467,175.348,17.339,152.619
C06691=1091.770,32.516,-57.451,175.347,17.338,152.619
C06692=1091.764,32.267,-57.436,175.345,17.336,152.619
C06693=1091.759,32.017,-57.421,175.343,17.335,152.619
C06694=1091.752,31.741,-57.404,175.341,17.334,152.619
C06695=1091.746,31.464,-57.388,175.339,17.332,152.619
C06696=1091.740,31.189,-57.371,175.338,17.330,152.619
C06697=1091.734,30.912,-57.354,175.335,17.329,152.620
C06698=1091.728,30.663,-57.340,175.334,17.327,152.619
C06699=1091.722,30.413,-57.324,175.331,17.326,152.620
C06700=1091.716,30.164,-57.310,175.330,17.324,152.620
C06701=1091.711,29.914,-57.294,175.327,17.323,152.620
C06702=1091.705,29.665,-57.279,175.326,17.321,152.620
C06703=1091.699,29.415,-57.264,175.324,17.320,152.620
C06704=1091.694,29.166,-57.249,175.322,17.318,152.620
C06705=1091.688,28.916,-57.234,175.320,17.317,152.620
C06706=1091.682,28.667,-57.219,175.319,17.316,152.620
C06707=1091.676,28.417,-57.204,175.316,17.314,152.620
C06708=1091.671,28.168,-57.189,175.315,17.313,152.620
C06709=1091.664,27.918,-57.174,175.313,17.311,152.620
C06710=1091.659,27.669,-57.159,175.311,17.310,152.620
C06711=1091.653,27.419,-57.144,175.309,17.309,152.620
C06712=1091.647,27.170,-57.130,175.307,17.306,152.620
C06713=1091.642,26.920,-57.115,175.305,17.305,152.621
C06714=1091.636,26.671,-57.100,175.304,17.304,152.621
C06715=1091.630,26.422,-57.085,175.301,17.302,152.621
C06716=1091.625,26.172,-57.070,175.300,17.301,152.621
C06717=1091.619,25.923,-57.055,175.298,17.300,152.621
C06718=1091.613,25.673,-57.041,175.296,17.298,152.621
C06719=1091.608,25.424,-57.026,175.295,17.297,152.621
C06720=1091.601,25.174,-57.011,175.293,17.295,152.621
C06721=1091.596,24.925,-56.996,175.290,17.294,152.621
C06722=1091.590,24.675,-56.981,175.289,17.293,152.621
C06723=1091.584,24.425,-56.967,175.287,17.291,152.621
C06724=1091.578,24.176,-56.952,175.285,17.289,152.621
C06725=1091.572,23.927,-56.937,175.283,17.288,152.621
C06726=1091.567,23.677,-56.922,175.282,17.287,152.621
C06727=1091.561,23.428,-56.907,175.280,17.285,152.622
C06728=1091.555,23.178,-56.893,175.278,17.284,152.622
C06729=1091.550,22.928,-56.878,175.277,17.282,152.622
C06730=1091.544,22.679,-56.863,175.274,17.281,152.622
C06731=1091.538,22.429,-56.849,175.272,17.280,152.622
C06732=1091.532,22.180,-56.834,175.271,17.278,152.622
C06733=1091.527,21.931,-56.819,175.269,17.276,152.622
C06734=1091.521,21.681,-56.804,175.267,17.275,152.622
C06735=1091.515,21.432,-56.791,175.266,17.274,152.622
C06736=1091.509,21.182,-56.776,175.263,17.272,152.622
C06737=1091.504,20.933,-56.760,175.262,17.270,152.622
C06738=1091.498,20.683,-56.747,175.260,17.269,152.622
C06739=1091.492,20.433,-56.732,175.258,17.267,152.622
C06740=1091.486,20.185,-56.717,175.256,17.266,152.622
C06741=1091.481,19.934,-56.702,175.255,17.265,152.622
C06742=1091.475,19.685,-56.688,175.252,17.263,152.622
C06743=1091.470,19.435,-56.674,175.251,17.261,152.622
C06744=1091.463,19.186,-56.659,175.249,17.260,152.622
C06745=1091.457,18.937,-56.644,175.247,17.259,152.623
C06746=1091.452,18.687,-56.630,175.246,17.257,152.623
C06747=1091.446,18.437,-56.615,175.244,17.256,152.623
C06748=1091.441,18.188,-56.601,175.241,17.254,152.623
C06749=1091.434,17.938,-56.586,175.240,17.253,152.623
C06750=1091.429,17.689,-56.571,175.238,17.252,152.623
C06751=1091.423,17.439,-56.558,175.236,17.249,152.623
C06752=1091.417,17.190,-56.543,175.235,17.248,152.623
C06753=1091.411,16.940,-56.529,175.233,17.247,152.623
C06754=1091.405,16.691,-56.514,175.231,17.245,152.623
C06755=1091.400,16.441,-56.499,175.229,17.244,152.623
C06756=1091.394,16.192,-56.485,175.228,17.243,152.623
C06757=1091.389,15.942,-56.471,175.225,17.241,152.623
C06758=1091.382,15.667,-56.455,175.224,17.240,152.623
C06759=1091.376,15.392,-56.439,175.222,17.237,152.623
C06760=1091.369,15.118,-56.423,175.220,17.236,152.623
C06761=1091.363,14.843,-56.407,175.218,17.234,152.623
C06762=1091.358,14.594,-56.393,175.216,17.233,152.623
C06763=1091.351,14.344,-56.378,175.215,17.232,152.624
C06764=1091.346,14.094,-56.364,175.212,17.230,152.624
C06765=1091.340,13.845,-56.350,175.211,17.229,152.624
C06766=1091.334,13.595,-56.336,175.209,17.228,152.624
C06767=1091.328,13.346,-56.321,175.207,17.225,152.624
C06768=1091.323,13.097,-56.307,175.205,17.224,152.624
C06769=1091.316,12.847,-56.292,175.204,17.223,152.624
C06770=1091.311,12.597,-56.278,175.202,17.222,152.624
C06771=1091.305,12.348,-56.264,175.200,17.220,152.624
C06772=1091.298,12.098,-56.250,175.199,17.218,152.624
C06773=1091.293,11.849,-56.236,175.197,17.217,152.624
C06774=1091.287,11.600,-56.222,175.194,17.216,152.624
C06775=1091.281,11.350,-56.207,175.193,17.214,152.624
C06776=1091.275,11.100,-56.194,175.191,17.213,152.624
C06777=1091.270,10.851,-56.179,175.190,17.212,152.624
C06778=1091.264,10.601,-56.165,175.188,17.210,152.624
C06779=1091.258,10.351,-56.151,175.186,17.208,152.624
C06780=1091.252,10.102,-56.136,175.185,17.207,152.624
C06781=1091.247,9.853,-56.122,175.182,17.205,152.625
C06782=1091.240,9.603,-56.108,175.181,17.204,152.625
C06783=1091.234,9.354,-56.094,175.179,17.202,152.625
C06784=1091.229,9.104,-56.080,175.177,17.201,152.625
C06785=1091.223,8.854,-56.066,175.175,17.199,152.625
C06786=1091.217,8.605,-56.052,175.174,17.198,152.625
C06787=1091.211,8.355,-56.038,175.172,17.197,152.625
C06788=1091.206,8.106,-56.024,175.170,17.195,152.625
C06789=1091.200,7.856,-56.009,175.168,17.194,152.625
C06790=1091.193,7.607,-55.996,175.167,17.192,152.625
C06791=1091.188,7.357,-55.982,175.165,17.190,152.625
C06792=1091.182,7.108,-55.968,175.163,17.189,152.625
C06793=1091.176,6.858,-55.953,175.162,17.188,152.625
C06794=1091.171,6.609,-55.939,175.160,17.187,152.625
C06795=1091.165,6.359,-55.925,175.158,17.184,152.625
C06796=1091.160,6.109,-55.911,175.156,17.183,152.625
C06797=1091.153,5.860,-55.898,175.155,17.182,152.625
C06798=1091.147,5.611,-55.883,175.153,17.181,152.625
C06799=1091.142,5.361,-55.869,175.151,17.179,152.625
C06800=1091.136,5.111,-55.855,175.149,17.177,152.625
C06801=1091.131,4.862,-55.841,175.148,17.176,152.626
C06802=1091.125,4.612,-55.828,175.146,17.174,152.626
C06803=1091.118,4.363,-55.813,175.144,17.173,152.626
C06804=1091.113,4.113,-55.799,175.143,17.171,152.626
C06805=1091.107,3.864,-55.786,175.141,17.170,152.626
C06806=1091.102,3.614,-55.772,175.139,17.168,152.626
C06807=1091.096,3.365,-55.758,175.137,17.167,152.626
C06808=1091.090,3.115,-55.745,175.136,17.165,152.626
C06809=1091.084,2.865,-55.730,175.134,17.164,152.626
C06810=1091.078,2.615,-55.716,175.132,17.162,152.626
C06811=1091.073,2.366,-55.702,175.130,17.161,152.626
C06812=1091.067,2.117,-55.688,175.129,17.160,152.626
C06813=1091.061,1.868,-55.675,175.127,17.158,152.626
C06814=1091.055,1.618,-55.661,175.125,17.157,152.626
C06815=1091.050,1.369,-55.647,175.124,17.155,152.626
C06816=1091.044,1.118,-55.633,175.122,17.154,152.626
C06817=1091.038,0.869,-55.620,175.120,17.152,152.626
C06818=1091.032,0.619,-55.606,175.118,17.151,152.626
C06819=1091.027,0.370,-55.592,175.117,17.149,152.626
C06820=1091.021,0.120,-55.578,175.115,17.148,152.626
C06821=1091.015,-0.129,-55.565,175.113,17.146,152.626
C06822=1091.009,-0.402,-55.549,175.111,17.145,152.626
C06823=1091.002,-0.675,-55.534,175.109,17.142,152.626
C06824=1090.997,-0.947,-55.519,175.108,17.141,152.626
C06825=1090.990,-1.221,-55.504,175.105,17.139,152.626
C06826=1090.984,-1.470,-55.490,175.104,17.138,152.626
C06827=1090.979,-1.720,-55.477,175.102,17.136,152.626
C06828=1090.973,-1.969,-55.463,175.101,17.135,152.626
C06829=1090.967,-2.218,-55.449,175.099,17.133,152.627
C06830=1090.962,-2.468,-55.436,175.097,17.132,152.627
C06831=1090.956,-2.718,-55.422,175.096,17.130,152.627
C06832=1090.950,-2.967,-55.408,175.094,17.129,152.627
C06833=1090.945,-3.216,-55.395,175.092,17.127,152.627
C06834=1090.939,-3.466,-55.381,175.090,17.126,152.627
C06835=1090.933,-3.715,-55.367,175.089,17.124,152.627
C06836=1090.927,-3.966,-55.353,175.087,17.123,152.627
C06837=1090.921,-4.215,-55.340,175.085,17.121,152.627
C06838=1090.916,-4.465,-55.327,175.083,17.120,152.627
C06839=1090.909,-4.714,-55.314,175.082,17.118,152.627
C06840=1090.904,-4.964,-55.300,175.080,17.117,152.627
C06841=1090.898,-5.213,-55.286,175.079,17.116,152.627
C06842=1090.892,-5.463,-55.273,175.077,17.114,152.627
C06843=1090.886,-5.712,-55.259,175.075,17.113,152.627
C06844=1090.880,-5.962,-55.245,175.074,17.111,152.627
C06845=1090.874,-6.212,-55.232,175.072,17.110,152.627
C06846=1090.868,-6.462,-55.219,175.070,17.108,152.627
C06847=1090.862,-6.711,-55.205,175.068,17.107,152.627
C06848=1090.857,-6.961,-55.191,175.067,17.105,152.627
C06849=1090.851,-7.210,-55.178,175.065,17.104,152.627
C06850=1090.845,-7.459,-55.164,175.063,17.102,152.627
C06851=1090.839,-7.709,-55.151,175.061,17.101,152.627
C06852=1090.834,-7.959,-55.138,175.060,17.099,152.627
C06853=1090.827,-8.208,-55.125,175.058,17.098,152.628
C06854=1090.822,-8.458,-55.111,175.057,17.097,152.627
C06855=1090.816,-8.707,-55.098,175.055,17.095,152.628
C06856=1090.811,-8.957,-55.084,175.053,17.094,152.628
C06857=1090.804,-9.206,-55.071,175.052,17.092,152.628
C06858=1090.798,-9.456,-55.058,175.050,17.091,152.628
C06859=1090.793,-9.705,-55.044,175.048,17.089,152.628
C06860=1090.787,-9.955,-55.031,175.046,17.088,152.628
C06861=1090.781,-10.205,-55.018,175.045,17.086,152.628
C06862=1090.775,-10.454,-55.004,175.043,17.085,152.628
C06863=1090.770,-10.704,-54.990,175.042,17.084,152.628
C06864=1090.764,-10.953,-54.978,175.039,17.082,152.628
C06865=1090.758,-11.203,-54.964,175.038,17.080,152.628
C06866=1090.752,-11.452,-54.951,175.036,17.079,152.628
C06867=1090.746,-11.702,-54.938,175.035,17.078,152.628
C06868=1090.741,-11.952,-54.924,175.033,17.076,152.628
C06869=1090.734,-12.201,-54.911,175.031,17.074,152.628
C06870=1090.729,-12.451,-54.898,175.030,17.073,152.628
C06871=1090.723,-12.700,-54.885,175.028,17.072,152.628
C06872=1090.717,-12.950,-54.871,175.027,17.070,152.628
C06873=1090.712,-13.200,-54.858,175.025,17.068,152.628
C06874=1090.705,-13.449,-54.845,175.023,17.067,152.628
C06875=1090.700,-13.699,-54.831,175.022,17.066,152.628
C06876=1090.694,-13.949,-54.819,175.020,17.064,152.628
C06877=1090.688,-14.198,-54.805,175.019,17.063,152.628
C06878=1090.683,-14.448,-54.792,175.016,17.061,152.628
C06879=1090.676,-14.697,-54.779,175.015,17.060,152.628
C06880=1090.671,-14.947,-54.765,175.013,17.058,152.629
C06881=1090.665,-15.197,-54.752,175.012,17.057,152.628
C06882=1090.659,-15.446,-54.739,175.010,17.056,152.629
C06883=1090.653,-15.696,-54.727,175.008,17.054,152.629
C06884=1090.647,-15.946,-54.713,175.006,17.052,152.629
C06885=1090.642,-16.195,-54.700,175.005,17.051,152.629
C06886=1090.635,-16.466,-54.686,175.003,17.050,152.629
C06887=1090.629,-16.738,-54.672,175.001,17.048,152.629
C06888=1090.622,-17.009,-54.658,175.000,17.046,152.629
C06889=1090.616,-17.280,-54.644,174.997,17.045,152.629
C06890=1090.610,-17.528,-54.631,174.996,17.043,152.629
C06891=1090.605,-17.779,-54.618,174.994,17.042,152.629
C06892=1090.599,-18.028,-54.604,174.993,17.040,152.629
C06893=1090.593,-18.278,-54.592,174.991,17.039,152.629
C06894=1090.587,-18.527,-54.578,174.990,17.038,152.629
C06895=1090.581,-18.777,-54.566,174.987,17.036,152.629
C06896=1090.575,-19.026,-54.552,174.986,17.035,152.629
C06897=1090.569,-19.276,-54.539,174.984,17.033,152.629
C06898=1090.563,-19.526,-54.526,174.983,17.032,152.629
C06899=1090.557,-19.775,-54.514,174.981,17.031,152.629
C06900=1090.551,-20.025,-54.500,174.979,17.029,152.629
C06901=1090.545,-20.275,-54.488,174.978,17.027,152.629
C06902=1090.540,-20.524,-54.474,174.976,17.026,152.629
C06903=1090.534,-20.773,-54.462,174.975,17.025,152.629
C06904=1090.528,-21.023,-54.449,174.973,17.024,152.630
C06905=1090.522,-21.273,-54.436,174.972,17.022,152.629
C06906=1090.516,-21.522,-54.423,174.969,17.020,152.630
C06907=1090.510,-21.772,-54.410,174.968,17.019,152.630
C06908=1090.505,-22.022,-54.397,174.966,17.018,152.630
C06909=1090.499,-22.272,-54.384,174.965,17.016,152.630
C06910=1090.493,-22.521,-54.371,174.963,17.015,152.630
C06911=1090.488,-22.770,-54.359,174.961,17.013,152.630
C06912=1090.482,-23.020,-54.346,174.959,17.012,152.630
C06913=1090.475,-23.269,-54.333,174.958,17.010,152.630
C06914=1090.469,-23.519,-54.321,174.956,17.009,152.630
C06915=1090.464,-23.769,-54.307,174.955,17.008,152.630
C06916=1090.458,-24.019,-54.294,174.953,17.006,152.630
C06917=1090.452,-24.269,-54.282,174.951,17.004,152.630
C06918=1090.447,-24.518,-54.269,174.950,17.003,152.630
C06919=1090.441,-24.767,-54.256,174.948,17.002,152.630
C06920=1090.435,-25.017,-54.244,174.947,17.000,152.630
C06921=1090.429,-25.267,-54.231,174.945,16.999,152.630
C06922=1090.423,-25.516,-54.218,174.944,16.997,152.630
C06923=1090.418,-25.766,-54.205,174.941,16.996,152.630
C06924=1090.412,-26.015,-54.192,174.940,16.995,152.630
C06925=1090.406,-26.265,-54.180,174.938,16.993,152.630
C06926=1090.400,-26.515,-54.167,174.937,16.992,152.630
C06927=1090.394,-26.764,-54.154,174.935,16.990,152.630
C06928=1090.389,-27.014,-54.142,174.934,16.989,152.631
C06929=1090.383,-27.264,-54.129,174.932,16.988,152.630
C06930=1090.377,-27.513,-54.116,174.930,16.986,152.631
C06931=1090.371,-27.763,-54.103,174.929,16.984,152.631
C06932=1090.365,-28.013,-54.091,174.927,16.983,152.631
C06933=1090.359,-28.262,-54.078,174.925,16.982,152.631
C06934=1090.353,-28.511,-54.065,174.924,16.980,152.631
C06935=1090.347,-28.761,-54.053,174.922,16.979,152.631
C06936=1090.341,-29.010,-54.041,174.921,16.978,152.631
C06937=1090.335,-29.260,-54.028,174.919,16.976,152.631
C06938=1090.329,-29.510,-54.016,174.917,16.975,152.631
C06939=1090.323,-29.760,-54.003,174.916,16.973,152.631
C06940=1090.317,-30.009,-53.990,174.914,16.972,152.631
C06941=1090.312,-30.259,-53.978,174.913,16.971,152.631
C06942=1090.306,-30.508,-53.965,174.911,16.969,152.631
C06943=1090.300,-30.758,-53.953,174.910,16.968,152.631
C06944=1090.294,-31.008,-53.940,174.907,16.966,152.631
C06945=1090.289,-31.257,-53.928,174.906,16.965,152.631
C06946=1090.283,-31.507,-53.915,174.904,16.963,152.631
C06947=1090.276,-31.756,-53.903,174.903,16.962,152.631
C06948=1090.270,-32.006,-53.890,174.901,16.961,152.631
C06949=1090.264,-32.255,-53.878,174.900,16.960,152.631
C06950=1090.258,-32.526,-53.864,174.897,16.958,152.632
C06951=1090.252,-32.797,-53.850,174.896,16.956,152.632
C06952=1090.245,-33.067,-53.837,174.894,16.955,152.632
C06953=1090.239,-33.337,-53.824,174.893,16.954,152.632
C06954=1090.233,-33.587,-53.811,174.890,16.952,152.632
C06955=1090.228,-33.836,-53.799,174.889,16.950,152.632
C06956=1090.221,-34.085,-53.787,174.887,16.949,152.632
C06957=1090.215,-34.335,-53.774,174.886,16.948,152.632
C06958=1090.209,-34.585,-53.762,174.884,16.947,152.632
C06959=1090.204,-34.834,-53.750,174.883,16.945,152.632
C06960=1090.198,-35.084,-53.737,174.881,16.944,152.632
C06961=1090.192,-35.334,-53.725,174.880,16.943,152.632
C06962=1090.187,-35.583,-53.712,174.878,16.941,152.632
C06963=1090.180,-35.833,-53.700,174.876,16.939,152.632
C06964=1090.174,-36.083,-53.688,174.874,16.938,152.632
C06965=1090.168,-36.333,-53.675,174.873,16.937,152.632
C06966=1090.163,-36.582,-53.663,174.871,16.936,152.632
C06967=1090.157,-36.832,-53.651,174.870,16.934,152.632
C06968=1090.151,-37.082,-53.638,174.868,16.933,152.632
C06969=1090.145,-37.331,-53.626,174.867,16.931,152.632
C06970=1090.139,-37.580,-53.614,174.865,16.930,152.632
C06971=1090.133,-37.830,-53.601,174.863,16.928,152.633
C06972=1090.128,-38.079,-53.589,174.862,16.927,152.632
C06973=1090.123,-38.330,-53.577,174.860,16.926,152.633
C06974=1090.116,-38.580,-53.565,174.859,16.924,152.633
C06975=1090.111,-38.829,-53.553,174.857,16.923,152.633
C06976=1090.105,-39.079,-53.541,174.855,16.922,152.633
C06977=1090.098,-39.328,-53.529,174.854,16.920,152.633
C06978=1090.093,-39.577,-53.516,174.852,16.919,152.633
C06979=1090.087,-39.827,-53.504,174.851,16.918,152.633
C06980=1090.080,-40.077,-53.492,174.849,16.916,152.633
C06981=1090.075,-40.326,-53.480,174.847,16.915,152.633
C06982=1090.069,-40.576,-53.467,174.845,16.914,152.633
C06983=1090.063,-40.826,-53.456,174.844,16.912,152.633
C06984=1090.057,-41.076,-53.443,174.842,16.911,152.633
C06985=1090.051,-41.325,-53.431,174.841,16.909,152.633
C06986=1090.045,-41.575,-53.419,174.839,16.908,152.633
C06987=1090.039,-41.825,-53.407,174.838,16.907,152.633
C06988=1090.033,-42.073,-53.395,174.836,16.905,152.633
C06989=1090.027,-42.324,-53.383,174.835,16.904,152.633
C06990=1090.021,-42.574,-53.371,174.833,16.903,152.633
C06991=1090.015,-42.823,-53.359,174.831,16.901,152.633
C06992=1090.009,-43.073,-53.347,174.829,16.900,152.634
C06993=1090.004,-43.322,-53.334,174.828,16.899,152.634
C06994=1089.998,-43.572,-53.323,174.826,16.897,152.634
C06995=1089.992,-43.822,-53.311,174.825,16.896,152.634
C06996=1089.986,-44.071,-53.299,174.823,16.895,152.634
C06997=1089.980,-44.321,-53.286,174.822,16.893,152.634
C06998=1089.974,-44.571,-53.274,174.820,16.892,152.634
C06999=1089.968,-44.820,-53.263,174.819,16.891,152.634
C07000=1089.962,-45.070,-53.250,174.817,16.890,152.634
C07001=1089.956,-45.319,-53.239,174.816,16.888,152.634
C07002=1089.951,-45.569,-53.227,174.814,16.887,152.634
C07003=1089.945,-45.819,-53.214,174.813,16.886,152.634
C07004=1089.939,-46.068,-53.203,174.810,16.884,152.634
C07005=1089.933,-46.318,-53.190,174.809,16.883,152.634
C07006=1089.927,-46.567,-53.179,174.807,16.881,152.634
C07007=1089.921,-46.817,-53.167,174.806,16.880,152.634
C07008=1089.914,-47.067,-53.155,174.804,16.879,152.635
C07009=1089.909,-47.317,-53.143,174.803,16.877,152.635
C07010=1089.903,-47.566,-53.132,174.801,16.876,152.635
C07011=1089.898,-47.815,-53.119,174.799,16.875,152.635
C07012=1089.892,-48.066,-53.108,174.798,16.874,152.635
C07013=1089.886,-48.315,-53.096,174.796,16.873,152.635
C07014=1089.880,-48.586,-53.083,174.795,16.871,152.635
C07015=1089.873,-48.856,-53.070,174.793,16.869,152.635
C07016=1089.866,-49.127,-53.057,174.791,16.868,152.635
C07017=1089.861,-49.398,-53.044,174.790,16.867,152.635
C07018=1089.854,-49.648,-53.032,174.788,16.865,152.635
C07019=1089.849,-49.897,-53.021,174.786,16.864,152.635
C07020=1089.842,-50.147,-53.009,174.785,16.863,152.635
C07021=1089.837,-50.396,-52.997,174.783,16.862,152.635
C07022=1089.831,-50.646,-52.986,174.782,16.860,152.635
C07023=1089.825,-50.895,-52.973,174.780,16.859,152.635
C07024=1089.819,-51.146,-52.962,174.779,16.858,152.635
C07025=1089.812,-51.395,-52.950,174.777,16.857,152.635
C07026=1089.806,-51.644,-52.939,174.775,16.856,152.636
C07027=1089.801,-51.895,-52.927,174.774,16.854,152.636
C07028=1089.795,-52.143,-52.915,174.772,16.852,152.636
C07029=1089.788,-52.394,-52.904,174.770,16.851,152.636
C07030=1089.782,-52.644,-52.891,174.768,16.850,152.636
C07031=1089.777,-52.893,-52.880,174.767,16.849,152.636
C07032=1089.770,-53.143,-52.868,174.765,16.848,152.636
C07033=1089.764,-53.392,-52.858,174.764,16.846,152.636
C07034=1089.758,-53.642,-52.845,174.762,16.845,152.636
C07035=1089.753,-53.891,-52.834,174.761,16.844,152.636
C07036=1089.746,-54.141,-52.822,174.759,16.843,152.636
C07037=1089.740,-54.392,-52.810,174.758,16.841,152.636
C07038=1089.734,-54.640,-52.799,174.756,16.840,152.636
C07039=1089.728,-54.891,-52.788,174.754,16.839,152.637
C07040=1089.722,-55.139,-52.776,174.753,16.838,152.637
C07041=1089.716,-55.390,-52.764,174.751,16.837,152.637
C07042=1089.710,-55.639,-52.752,174.750,16.835,152.637
C07043=1089.704,-55.889,-52.741,174.748,16.834,152.637
C07044=1089.698,-56.138,-52.730,174.746,16.833,152.637
C07045=1089.692,-56.388,-52.718,174.745,16.832,152.637
C07046=1089.686,-56.637,-52.706,174.743,16.831,152.637
C07047=1089.680,-56.887,-52.695,174.742,16.829,152.637
C07048=1089.674,-57.136,-52.683,174.740,16.828,152.637
C07049=1089.668,-57.387,-52.672,174.739,16.827,152.637
C07050=1089.663,-57.636,-52.661,174.737,16.826,152.637
C07051=1089.656,-57.886,-52.649,174.735,16.825,152.638
C07052=1089.650,-58.135,-52.638,174.734,16.823,152.637
C07053=1089.644,-58.385,-52.626,174.732,16.822,152.638
C07054=1089.639,-58.635,-52.614,174.731,16.821,152.638
C07055=1089.632,-58.885,-52.603,174.729,16.820,152.638
C07056=1089.626,-59.134,-52.592,174.728,16.819,152.638
C07057=1089.620,-59.384,-52.580,174.726,16.817,152.638
C07058=1089.614,-59.634,-52.569,174.725,16.816,152.638
C07059=1089.608,-59.883,-52.557,174.723,16.815,152.638
C07060=1089.602,-60.133,-52.546,174.721,16.814,152.638
C07061=1089.596,-60.383,-52.535,174.720,16.813,152.638
C07062=1089.590,-60.632,-52.523,174.718,16.811,152.638
C07063=1089.584,-60.882,-52.512,174.717,16.810,152.638
C07064=1089.579,-61.132,-52.500,174.715,16.809,152.638
C07065=1089.573,-61.381,-52.489,174.713,16.808,152.639
C07066=1089.566,-61.631,-52.478,174.712,16.806,152.639
C07067=1089.561,-61.880,-52.467,174.710,16.805,152.639
C07068=1089.554,-62.130,-52.455,174.709,16.804,152.639
C07069=1089.548,-62.380,-52.444,174.707,16.803,152.639
C07070=1089.543,-62.630,-52.432,174.706,16.802,152.639
C07071=1089.537,-62.880,-52.421,174.704,16.800,152.639
C07072=1089.531,-63.128,-52.410,174.702,16.799,152.639
C07073=1089.524,-63.379,-52.398,174.701,16.798,152.639
C07074=1089.519,-63.628,-52.387,174.699,16.797,152.639
C07075=1089.512,-63.878,-52.376,174.698,16.795,152.639
C07076=1089.507,-64.127,-52.364,174.696,16.794,152.639
C07077=1089.501,-64.377,-52.353,174.694,16.793,152.640
C07078=1089.495,-64.649,-52.341,174.693,16.792,152.640
C07079=1089.489,-64.921,-52.329,174.691,16.791,152.640
C07080=1089.482,-65.193,-52.317,174.690,16.789,152.640
C07081=1089.475,-65.465,-52.305,174.687,16.788,152.640
C07082=1089.469,-65.715,-52.293,174.686,16.787,152.640
C07083=1089.463,-65.964,-52.281,174.685,16.786,152.640
C07084=1089.458,-66.214,-52.270,174.683,16.785,152.640
C07085=1089.451,-66.464,-52.259,174.682,16.783,152.640
C07086=1089.446,-66.714,-52.248,174.680,16.782,152.640
C07087=1089.440,-66.963,-52.237,174.679,16.781,152.640
C07088=1089.434,-67.213,-52.226,174.677,16.780,152.640
C07089=1089.427,-67.462,-52.215,174.675,16.779,152.641
C07090=1089.422,-67.712,-52.204,174.674,16.778,152.641
C07091=1089.415,-67.962,-52.192,174.672,16.777,152.641
C07092=1089.410,-68.212,-52.181,174.671,16.775,152.641
C07093=1089.405,-68.461,-52.170,174.669,16.774,152.641
C07094=1089.398,-68.711,-52.159,174.668,16.773,152.641
C07095=1089.393,-68.961,-52.148,174.666,16.772,152.641
C07096=1089.387,-69.210,-52.137,174.664,16.771,152.641
C07097=1089.380,-69.461,-52.126,174.663,16.769,152.641
C07098=1089.375,-69.710,-52.115,174.661,16.768,152.641
C07099=1089.369,-69.959,-52.103,174.660,16.767,152.641
C07100=1089.362,-70.209,-52.092,174.658,16.766,152.641
C07101=1089.357,-70.459,-52.081,174.657,16.765,152.642
C07102=1089.351,-70.708,-52.070,174.655,16.763,152.642
C07103=1089.345,-70.958,-52.059,174.653,16.762,152.642
C07104=1089.339,-71.208,-52.048,174.652,16.761,152.642
C07105=1089.334,-71.458,-52.037,174.650,16.760,152.642
C07106=1089.328,-71.707,-52.026,174.649,16.758,152.642
C07107=1089.322,-71.957,-52.015,174.647,16.757,152.642
C07108=1089.316,-72.207,-52.004,174.646,16.757,152.642
C07109=1089.310,-72.456,-51.993,174.645,16.756,152.642
C07110=1089.304,-72.706,-51.982,174.643,16.755,152.642
C07111=1089.298,-72.956,-51.971,174.641,16.753,152.642
C07112=1089.292,-73.205,-51.960,174.640,16.752,152.643
C07113=1089.287,-73.455,-51.949,174.638,16.751,152.643
C07114=1089.281,-73.704,-51.938,174.636,16.750,152.643
C07115=1089.275,-73.955,-51.927,174.635,16.749,152.643
C07116=1089.269,-74.204,-51.916,174.633,16.747,152.643
C07117=1089.263,-74.454,-51.905,174.632,16.746,152.643
C07118=1089.257,-74.703,-51.894,174.630,16.745,152.643
C07119=1089.251,-74.953,-51.883,174.629,16.744,152.643
C07120=1089.245,-75.202,-51.873,174.627,16.743,152.643
C07121=1089.239,-75.452,-51.862,174.625,16.742,152.643
C07122=1089.233,-75.703,-51.851,174.625,16.741,152.643
C07123=1089.227,-75.952,-51.840,174.623,16.740,152.643
C07124=1089.221,-76.202,-51.830,174.621,16.739,152.644
C07125=1089.216,-76.451,-51.819,174.620,16.738,152.644
C07126=1089.209,-76.701,-51.807,174.618,16.737,152.644
C07127=1089.203,-76.951,-51.797,174.616,16.736,152.644
C07128=1089.197,-77.200,-51.786,174.615,16.735,152.644
C07129=1089.191,-77.450,-51.775,174.613,16.734,152.644
C07130=1089.185,-77.700,-51.764,174.611,16.732,152.644
C07131=1089.179,-77.949,-51.753,174.610,16.731,152.644
C07132=1089.174,-78.199,-51.743,174.608,16.730,152.644
C07133=1089.167,-78.449,-51.732,174.607,16.729,152.645
C07134=1089.161,-78.699,-51.722,174.606,16.729,152.645
C07135=1089.155,-78.948,-51.711,174.604,16.727,152.645
C07136=1089.149,-79.198,-51.700,174.603,16.726,152.645
C07137=1089.144,-79.447,-51.689,174.601,16.725,152.645
C07138=1089.137,-79.697,-51.678,174.599,16.724,152.645
C07139=1089.131,-79.947,-51.668,174.598,16.723,152.645
C07140=1089.125,-80.197,-51.657,174.596,16.722,152.645
C07141=1089.120,-80.446,-51.646,174.594,16.721,152.646
C07142=1089.112,-80.721,-51.635,174.592,16.720,152.646
C07143=1089.106,-80.994,-51.623,174.591,16.719,152.646
C07144=1089.099,-81.269,-51.612,174.589,16.718,152.646
C07145=1089.092,-81.543,-51.599,174.588,16.717,152.646
C07146=1089.086,-81.792,-51.590,174.586,16.716,152.646
C07147=1089.080,-82.043,-51.579,174.584,16.715,152.646
C07148=1089.074,-82.292,-51.568,174.583,16.713,152.646
C07149=1089.068,-82.541,-51.557,174.581,16.712,152.646
C07150=1089.062,-82.791,-51.547,174.580,16.712,152.647
C07151=1089.056,-83.042,-51.536,174.578,16.711,152.647
C07152=1089.049,-83.291,-51.526,174.577,16.710,152.647
C07153=1089.044,-83.540,-51.515,174.575,16.709,152.647
C07154=1089.038,-83.790,-51.505,174.573,16.708,152.647
C07155=1089.031,-84.040,-51.494,174.572,16.707,152.647
C07156=1089.025,-84.290,-51.483,174.570,16.706,152.647
C07157=1089.019,-84.539,-51.473,174.569,16.705,152.647
C07158=1089.014,-84.789,-51.463,174.567,16.705,152.648
C07159=1089.008,-85.038,-51.452,174.566,16.703,152.648
C07160=1089.001,-85.288,-51.441,174.564,16.702,152.648
C07161=1088.995,-85.538,-51.431,174.563,16.701,152.648
C07162=1088.989,-85.788,-51.421,174.561,16.700,152.648
C07163=1088.983,-86.037,-51.410,174.559,16.699,152.648
C07164=1088.978,-86.287,-51.400,174.558,16.698,152.648
C07165=1088.971,-86.537,-51.389,174.557,16.698,152.649
C07166=1088.965,-86.787,-51.378,174.555,16.697,152.649
C07167=1088.959,-87.036,-51.369,174.553,16.696,152.649
C07168=1088.953,-87.286,-51.358,174.552,16.694,152.649
C07169=1088.946,-87.535,-51.347,174.550,16.693,152.649
C07170=1088.940,-87.786,-51.337,174.548,16.692,152.649
C07171=1088.935,-88.035,-51.326,174.547,16.691,152.649
C07172=1088.928,-88.285,-51.316,174.546,16.691,152.649
C07173=1088.923,-88.535,-51.306,174.544,16.690,152.649
C07174=1088.916,-88.784,-51.295,174.542,16.689,152.650
C07175=1088.911,-89.034,-51.285,174.541,16.688,152.650
C07176=1088.904,-89.283,-51.275,174.539,16.687,152.650
C07177=1088.898,-89.533,-51.264,174.537,16.686,152.650
C07178=1088.893,-89.783,-51.253,174.536,16.685,152.650
C07179=1088.886,-90.033,-51.243,174.535,16.684,152.650
C07180=1088.881,-90.283,-51.233,174.533,16.683,152.650
C07181=1088.874,-90.532,-51.223,174.532,16.682,152.650
C07182=1088.869,-90.782,-51.213,174.530,16.681,152.651
C07183=1088.862,-91.031,-51.202,174.528,16.680,152.651
C07184=1088.856,-91.281,-51.191,174.526,16.679,152.651
C07185=1088.850,-91.531,-51.182,174.526,16.679,152.651
C07186=1088.844,-91.781,-51.171,174.524,16.678,152.651
C07187=1088.838,-92.030,-51.161,174.522,16.677,152.651
C07188=1088.832,-92.280,-51.150,174.520,16.676,152.652
C07189=1088.826,-92.530,-51.141,174.519,16.675,152.652
C07190=1088.820,-92.779,-51.130,174.518,16.674,152.652
C07191=1088.814,-93.029,-51.120,174.516,16.673,152.652
C07192=1088.808,-93.278,-51.109,174.515,16.672,152.652
C07193=1088.803,-93.529,-51.099,174.513,16.671,152.652
C07194=1088.796,-93.778,-51.089,174.511,16.670,152.652
C07195=1088.790,-94.029,-51.078,174.510,16.669,152.652
C07196=1088.784,-94.278,-51.068,174.509,16.669,152.652
C07197=1088.778,-94.528,-51.058,174.507,16.668,152.653
C07198=1088.772,-94.778,-51.048,174.505,16.667,152.653
C07199=1088.767,-95.027,-51.037,174.504,16.666,152.653
C07200=1088.760,-95.277,-51.028,174.502,16.665,152.653
C07201=1088.754,-95.526,-51.018,174.500,16.664,152.653
C07202=1088.748,-95.776,-51.007,174.499,16.664,152.653
C07203=1088.742,-96.025,-50.997,174.498,16.663,152.653
C07204=1088.737,-96.276,-50.987,174.496,16.661,152.654
C07205=1088.730,-96.525,-50.977,174.494,16.661,152.654
C07206=1088.724,-96.802,-50.966,174.492,16.660,152.654
C07207=1088.717,-97.078,-50.954,174.491,16.659,152.654
C07208=1088.711,-97.354,-50.943,174.489,16.657,152.654
C07209=1088.704,-97.631,-50.932,174.487,16.657,152.654
C07210=1088.698,-97.881,-50.922,174.486,16.656,152.655
C07211=1088.692,-98.130,-50.912,174.485,16.655,152.655
C07212=1088.686,-98.380,-50.902,174.483,16.655,152.655
C07213=1088.680,-98.630,-50.892,174.481,16.653,152.655
C07214=1088.673,-98.879,-50.882,174.480,16.652,152.655
C07215=1088.668,-99.130,-50.871,174.479,16.652,152.655
C07216=1088.662,-99.379,-50.862,174.477,16.651,152.655
C07217=1088.655,-99.629,-50.852,174.475,16.650,152.656
C07218=1088.649,-99.878,-50.842,174.473,16.650,152.656
C07219=1088.643,-100.128,-50.832,174.472,16.648,152.656
C07220=1088.637,-100.378,-50.822,174.471,16.648,152.656
C07221=1088.631,-100.627,-50.812,174.469,16.647,152.656
C07222=1088.625,-100.878,-50.802,174.467,16.646,152.656
C07223=1088.619,-101.127,-50.792,174.465,16.646,152.657
C07224=1088.613,-101.377,-50.782,174.464,16.644,152.657
C07225=1088.607,-101.626,-50.772,174.463,16.644,152.657
C07226=1088.601,-101.876,-50.762,174.461,16.643,152.657
C07227=1088.595,-102.126,-50.752,174.459,16.642,152.657
C07228=1088.588,-102.375,-50.742,174.458,16.642,152.657
C07229=1088.583,-102.626,-50.732,174.457,16.641,152.658
C07230=1088.577,-102.875,-50.722,174.455,16.640,152.658
C07231=1088.570,-103.125,-50.712,174.453,16.639,152.658
C07232=1088.564,-103.374,-50.703,174.452,16.638,152.658
C07233=1088.559,-103.624,-50.693,174.450,16.638,152.658
C07234=1088.552,-103.874,-50.682,174.449,16.637,152.658
C07235=1088.546,-104.123,-50.673,174.447,16.636,152.658
C07236=1088.540,-104.373,-50.663,174.445,16.635,152.659
C07237=1088.534,-104.623,-50.654,174.444,16.635,152.659
C07238=1088.528,-104.872,-50.643,174.443,16.634,152.659
C07239=1088.522,-105.122,-50.633,174.441,16.633,152.659
C07240=1088.516,-105.372,-50.624,174.439,16.632,152.659
C07241=1088.510,-105.622,-50.614,174.438,16.632,152.659
C07242=1088.504,-105.872,-50.604,174.437,16.631,152.660
C07243=1088.498,-106.121,-50.594,174.435,16.630,152.660
C07244=1088.491,-106.371,-50.584,174.433,16.629,152.660
C07245=1088.485,-106.621,-50.575,174.432,16.629,152.660
C07246=1088.479,-106.871,-50.565,174.430,16.628,152.660
C07247=1088.474,-107.121,-50.555,174.428,16.627,152.661
C07248=1088.468,-107.370,-50.545,174.427,16.626,152.661
C07249=1088.461,-107.620,-50.535,174.426,16.626,152.661
C07250=1088.455,-107.869,-50.525,174.424,16.625,152.661
C07251=1088.449,-108.119,-50.516,174.422,16.625,152.661
C07252=1088.443,-108.369,-50.506,174.420,16.623,152.661
C07253=1088.436,-108.619,-50.497,174.419,16.623,152.662
C07254=1088.430,-108.869,-50.487,174.418,16.622,152.662
C07255=1088.424,-109.118,-50.478,174.416,16.622,152.662
C07256=1088.419,-109.369,-50.467,174.414,16.621,152.662
C07257=1088.412,-109.618,-50.457,174.413,16.621,152.662
C07258=1088.406,-109.868,-50.448,174.411,16.619,152.662
C07259=1088.400,-110.117,-50.438,174.410,16.619,152.663
C07260=1088.394,-110.367,-50.428,174.409,16.618,152.663
C07261=1088.387,-110.617,-50.419,174.407,16.618,152.663
C07262=1088.381,-110.867,-50.409,174.405,16.617,152.663
C07263=1088.375,-111.117,-50.400,174.403,16.616,152.663
C07264=1088.370,-111.366,-50.390,174.402,16.615,152.663
C07265=1088.363,-111.615,-50.381,174.401,16.615,152.664
C07266=1088.357,-111.865,-50.371,174.399,16.614,152.664
C07267=1088.351,-112.115,-50.362,174.397,16.613,152.664
C07268=1088.345,-112.365,-50.352,174.396,16.613,152.664
C07269=1088.339,-112.615,-50.343,174.394,16.612,152.664
C07270=1088.332,-112.885,-50.332,174.392,16.611,152.665
C07271=1088.325,-113.156,-50.321,174.390,16.611,152.665
